LIN {X 0,Y 480.316,Z 788.973,A -85,B 0,C 180,E1 7511.477,E2 7511.477} C_VEL
LIN {X 0,Y 481.888,Z 749.339,A -85,B 0,C 180,E1 7512.908,E2 7512.908} C_VEL
LIN {X 0,Y 449.961,Z 691.44,A -85,B 0,C 180,E1 7518.516,E2 7518.516} C_VEL
LIN {X 0,Y 450.056,Z 691.44,A -85,B 0,C 180,E1 7529.299,E2 7529.299} C_VEL
LIN {X 0,Y 450.366,Z 691.44,A -85,B 0,C 180,E1 7539.308,E2 7539.308} C_VEL
LIN {X 0,Y 450.688,Z 691.44,A -85,B 0,C 180,E1 7549.353,E2 7549.353} C_VEL
LIN {X 0,Y 451.015,Z 691.44,A -85,B 0,C 180,E1 7559.059,E2 7559.059} C_VEL
LIN {X 0,Y 450.905,Z 691.44,A -85,B 0,C 180,E1 7569.708,E2 7569.708} C_VEL
LIN {X 0,Y 451.272,Z 693.873,A -85,B 0,C 180,E1 7570.495,E2 7570.495} C_VEL
LIN {X 0,Y 478.579,Z 746.673,A -85,B 0,C 180,E1 7575.537,E2 7575.537} C_VEL
LIN {X 0,Y 481.013,Z 759.563,A -85,B 0,C 180,E1 7576.393,E2 7576.393} C_VEL
LIN {X 0,Y 473.42,Z 824.079,A -85,B 0,C 180,E1 7580.014,E2 7580.014} C_VEL
LIN {X 0,Y 464.828,Z 880.115,A -85,B 0,C 180,E1 7585.277,E2 7585.277} C_VEL
LIN {X 0,Y 457.425,Z 928.806,A -85,B 0,C 180,E1 7592.429,E2 7592.429} C_VEL
LIN {X 0,Y 453.01,Z 964.235,A -85,B 0,C 180,E1 7600.513,E2 7600.513} C_VEL
LIN {X 0,Y 451.297,Z 983.991,A -85,B 0,C 180,E1 7608.117,E2 7608.117} C_VEL
LIN {X 0,Y 450.543,Z 992.725,A -85,B 0,C 180,E1 7616.237,E2 7616.237} C_VEL
LIN {X 0,Y 451.09,Z 989.426,A -85,B 0,C 180,E1 7624.147,E2 7624.147} C_VEL
LIN {X 0,Y 452.471,Z 971.841,A -85,B 0,C 180,E1 7632.949,E2 7632.949} C_VEL
LIN {X 0,Y 455.599,Z 939.796,A -85,B 0,C 180,E1 7641.38,E2 7641.38} C_VEL
LIN {X 0,Y 462.546,Z 894.419,A -85,B 0,C 180,E1 7648.826,E2 7648.826} C_VEL
LIN {X 0,Y 471.111,Z 840.184,A -85,B 0,C 180,E1 7654.62,E2 7654.62} C_VEL
LIN {X 0,Y 479.119,Z 776.379,A -85,B 0,C 180,E1 7658.798,E2 7658.798} C_VEL
LIN {X 0,Y 480.222,Z 748.401,A -85,B 0,C 180,E1 7660.124,E2 7660.124} C_VEL
LIN {X 0,Y 450.704,Z 691.44,A -85,B 0,C 180,E1 7665.682,E2 7665.682} C_VEL
LIN {X 0,Y 450.338,Z 691.44,A -85,B 0,C 180,E1 7674.914,E2 7674.914} C_VEL
LIN {X 0,Y 449.921,Z 691.44,A -85,B 0,C 180,E1 7684.252,E2 7684.252} C_VEL
LIN {X 0,Y 449.961,Z 691.44,A -85,B 0,C 180,E1 7693.743,E2 7693.743} C_VEL
LIN {X 0,Y 449.854,Z 691.44,A -85,B 0,C 180,E1 7703.8,E2 7703.8} C_VEL
LIN {X 0,Y 450.191,Z 691.44,A -85,B 0,C 180,E1 7713.295,E2 7713.295} C_VEL
LIN {X 0,Y 450.987,Z 691.44,A -85,B 0,C 180,E1 7725.362,E2 7725.362} C_VEL
LIN {X 0,Y 451.028,Z 691.44,A -85,B 0,C 180,E1 7735.153,E2 7735.153} C_VEL
LIN {X 0,Y 451.105,Z 691.44,A -85,B 0,C 180,E1 7742.869,E2 7742.869} C_VEL
LIN {X 0,Y 450.691,Z 691.44,A -85,B 0,C 180,E1 7752.617,E2 7752.617} C_VEL
LIN {X 0,Y 450.376,Z 691.44,A -85,B 0,C 180,E1 7762.769,E2 7762.769} C_VEL
LIN {X 0,Y 450.042,Z 691.44,A -85,B 0,C 180,E1 7771.477,E2 7771.477} C_VEL
LIN {X 0,Y 450.162,Z 693.331,A -85,B 0,C 180,E1 7781.862,E2 7781.862} C_VEL
LIN {X 0,Y 483.134,Z 752.334,A -85,B 0,C 180,E1 7787.26,E2 7787.26} C_VEL
LIN {X 0,Y 477.738,Z 816.415,A -85,B 0,C 180,E1 7789.779,E2 7789.779} C_VEL
LIN {X 0,Y 469.365,Z 878.521,A -85,B 0,C 180,E1 7794.164,E2 7794.164} C_VEL
LIN {X 0,Y 468.241,Z 886.122,A -85,B 0,C 180,E1 7794.871,E2 7794.871} C_VEL
LIN {X 0,Y 457.024,Z 913.577,A -85,B 0,C 180,E1 7797.294,E2 7797.294} C_VEL
LIN {X 0,Y 449.765,Z 960.326,A -85,B 0,C 180,E1 7804.307,E2 7804.307} C_VEL
LIN {X 0,Y 445.009,Z 995.719,A -85,B 0,C 180,E1 7812.691,E2 7812.691} C_VEL
LIN {X 0,Y 443.149,Z 1015.884,A -85,B 0,C 180,E1 7821.134,E2 7821.134} C_VEL
LIN {X 0,Y 442.869,Z 1022.836,A -85,B 0,C 180,E1 7829.017,E2 7829.017} C_VEL
LIN {X 0,Y 443.349,Z 1018.684,A -85,B 0,C 180,E1 7836.88,E2 7836.88} C_VEL
LIN {X 0,Y 444.601,Z 1000.182,A -85,B 0,C 180,E1 7845.846,E2 7845.846} C_VEL
LIN {X 0,Y 448.349,Z 967.674,A -85,B 0,C 180,E1 7854.28,E2 7854.28} C_VEL
LIN {X 0,Y 455.186,Z 924.286,A -85,B 0,C 180,E1 7861.341,E2 7861.341} C_VEL
LIN {X 0,Y 464.152,Z 867.494,A -85,B 0,C 180,E1 7867.331,E2 7867.331} C_VEL
LIN {X 0,Y 472.707,Z 801.444,A -85,B 0,C 180,E1 7871.569,E2 7871.569} C_VEL
LIN {X 0,Y 475.718,Z 752.484,A -85,B 0,C 180,E1 7873.469,E2 7873.469} C_VEL
LIN {X 0,Y 443.691,Z 696.419,A -85,B 0,C 180,E1 7878.995,E2 7878.995} C_VEL
LIN {X 0,Y 441.936,Z 691.44,A -85,B 0,C 180,E1 7879.576,E2 7879.576} C_VEL
LIN {X 0,Y 442.035,Z 691.44,A -85,B 0,C 180,E1 7890.179,E2 7890.179} C_VEL
LIN {X 0,Y 442.406,Z 691.44,A -85,B 0,C 180,E1 7901.01,E2 7901.01} C_VEL
LIN {X 0,Y 442.802,Z 691.44,A -85,B 0,C 180,E1 7911.153,E2 7911.153} C_VEL
LIN {X 0,Y 443.542,Z 691.44,A -85,B 0,C 180,E1 7921.003,E2 7921.003} C_VEL
LIN {X 0,Y 443.012,Z 692.481,A -85,B 0,C 180,E1 7929.261,E2 7929.261} C_VEL
LIN {X 0,Y 471.363,Z 747.296,A -85,B 0,C 180,E1 7934.765,E2 7934.765} C_VEL
LIN {X 0,Y 474.779,Z 761.729,A -85,B 0,C 180,E1 7935.841,E2 7935.841} C_VEL
LIN {X 0,Y 466.841,Z 825.244,A -85,B 0,C 180,E1 7939.475,E2 7939.475} C_VEL
LIN {X 0,Y 457.627,Z 881.883,A -85,B 0,C 180,E1 7944.912,E2 7944.912} C_VEL
LIN {X 0,Y 450.08,Z 928.17,A -85,B 0,C 180,E1 7951.859,E2 7951.859} C_VEL
LIN {X 0,Y 445.374,Z 963.375,A -85,B 0,C 180,E1 7959.945,E2 7959.945} C_VEL
LIN {X 0,Y 443.29,Z 984.327,A -85,B 0,C 180,E1 7968.121,E2 7968.121} C_VEL
LIN {X 0,Y 442.576,Z 992.432,A -85,B 0,C 180,E1 7975.544,E2 7975.544} C_VEL
LIN {X 0,Y 442.986,Z 990.028,A -85,B 0,C 180,E1 7983.678,E2 7983.678} C_VEL
LIN {X 0,Y 444.322,Z 974.867,A -85,B 0,C 180,E1 7992.099,E2 7992.099} C_VEL
LIN {X 0,Y 447.531,Z 944.098,A -85,B 0,C 180,E1 8000.863,E2 8000.863} C_VEL
LIN {X 0,Y 454.538,Z 900.358,A -85,B 0,C 180,E1 8008.566,E2 8008.566} C_VEL
LIN {X 0,Y 463.52,Z 846.298,A -85,B 0,C 180,E1 8014.696,E2 8014.696} C_VEL
LIN {X 0,Y 471.971,Z 784.847,A -85,B 0,C 180,E1 8019.019,E2 8019.019} C_VEL
LIN {X 0,Y 474.063,Z 751.552,A -85,B 0,C 180,E1 8020.649,E2 8020.649} C_VEL
LIN {X 0,Y 444.766,Z 696.762,A -85,B 0,C 180,E1 8026.198,E2 8026.198} C_VEL
LIN {X 0,Y 442.62,Z 691.44,A -85,B 0,C 180,E1 8026.945,E2 8026.945} C_VEL
LIN {X 0,Y 442.17,Z 691.44,A -85,B 0,C 180,E1 8037.604,E2 8037.604} C_VEL
LIN {X 0,Y 441.876,Z 691.44,A -85,B 0,C 180,E1 8046.944,E2 8046.944} C_VEL
LIN {X 0,Y 441.865,Z 691.44,A -85,B 0,C 180,E1 8057.598,E2 8057.598} C_VEL
LIN {X 0,Y 441.942,Z 691.44,A -85,B 0,C 180,E1 8067.824,E2 8067.824} C_VEL
LIN {X 0,Y 441.943,Z 691.44,A -85,B 0,C 180,E1 8076.722,E2 8076.722} C_VEL
LIN {X 0,Y 442.985,Z 691.44,A -85,B 0,C 180,E1 8087.522,E2 8087.522} C_VEL
LIN {X 0,Y 442.874,Z 691.44,A -85,B 0,C 180,E1 8097.032,E2 8097.032} C_VEL
LIN {X 0,Y 442.823,Z 691.44,A -85,B 0,C 180,E1 8104.891,E2 8104.891} C_VEL
LIN {X 0,Y 442.651,Z 691.44,A -85,B 0,C 180,E1 8114.873,E2 8114.873} C_VEL
LIN {X 0,Y 442.244,Z 691.44,A -85,B 0,C 180,E1 8125.369,E2 8125.369} C_VEL
LIN {X 0,Y 441.864,Z 691.44,A -85,B 0,C 180,E1 8136.184,E2 8136.184} C_VEL
LIN {X 0,Y 442.068,Z 692.886,A -85,B 0,C 180,E1 8140.727,E2 8140.727} C_VEL
LIN {X 0,Y 477.127,Z 755.611,A -85,B 0,C 180,E1 8146.717,E2 8146.717} C_VEL
LIN {X 0,Y 470.984,Z 819.692,A -85,B 0,C 180,E1 8149.346,E2 8149.346} C_VEL
LIN {X 0,Y 462.201,Z 881.081,A -85,B 0,C 180,E1 8153.828,E2 8153.828} C_VEL
LIN {X 0,Y 457.024,Z 913.577,A -85,B 0,C 180,E1 8157.294,E2 8157.294} C_VEL
LIN {X 0,Y 445.427,Z 938.536,A -85,B 0,C 180,E1 8160.146,E2 8160.146} C_VEL
LIN {X 0,Y 438.993,Z 978.351,A -85,B 0,C 180,E1 8167.649,E2 8167.649} C_VEL
LIN {X 0,Y 435.805,Z 1004.335,A -85,B 0,C 180,E1 8175.376,E2 8175.376} C_VEL
LIN {X 0,Y 435.111,Z 1019.184,A -85,B 0,C 180,E1 8183.405,E2 8183.405} C_VEL
LIN {X 0,Y 435.328,Z 1022.837,A -85,B 0,C 180,E1 8190.998,E2 8190.998} C_VEL
LIN {X 0,Y 435.348,Z 1015.887,A -85,B 0,C 180,E1 8199.024,E2 8199.024} C_VEL
LIN {X 0,Y 436.853,Z 995.72,A -85,B 0,C 180,E1 8207.642,E2 8207.642} C_VEL
LIN {X 0,Y 441.383,Z 962.92,A -85,B 0,C 180,E1 8215.667,E2 8215.667} C_VEL
LIN {X 0,Y 449.416,Z 915.357,A -85,B 0,C 180,E1 8222.997,E2 8222.997} C_VEL
LIN {X 0,Y 459.194,Z 856.838,A -85,B 0,C 180,E1 8228.769,E2 8228.769} C_VEL
LIN {X 0,Y 467.619,Z 792.407,A -85,B 0,C 180,E1 8232.591,E2 8232.591} C_VEL
LIN {X 0,Y 469.538,Z 755.476,A -85,B 0,C 180,E1 8234.06,E2 8234.06} C_VEL
LIN {X 0,Y 437.3,Z 697.979,A -85,B 0,C 180,E1 8239.937,E2 8239.937} C_VEL
LIN {X 0,Y 433.861,Z 691.44,A -85,B 0,C 180,E1 8240.866,E2 8240.866} C_VEL
LIN {X 0,Y 434.008,Z 691.44,A -85,B 0,C 180,E1 8251.866,E2 8251.866} C_VEL
LIN {X 0,Y 434.438,Z 691.44,A -85,B 0,C 180,E1 8262.756,E2 8262.756} C_VEL
LIN {X 0,Y 435.03,Z 691.44,A -85,B 0,C 180,E1 8273.826,E2 8273.826} C_VEL
LIN {X 0,Y 435.092,Z 691.44,A -85,B 0,C 180,E1 8283.021,E2 8283.021} C_VEL
LIN {X 0,Y 435.012,Z 692.594,A -85,B 0,C 180,E1 8288.011,E2 8288.011} C_VEL
LIN {X 0,Y 463.641,Z 746.298,A -85,B 0,C 180,E1 8293.815,E2 8293.815} C_VEL
LIN {X 0,Y 468.572,Z 764.043,A -85,B 0,C 180,E1 8295.283,E2 8295.283} C_VEL
LIN {X 0,Y 460.152,Z 827.524,A -85,B 0,C 180,E1 8299.004,E2 8299.004} C_VEL
LIN {X 0,Y 450.443,Z 883.623,A -85,B 0,C 180,E1 8304.532,E2 8304.532} C_VEL
LIN {X 0,Y 442.524,Z 928.985,A -85,B 0,C 180,E1 8311.512,E2 8311.512} C_VEL
LIN {X 0,Y 437.377,Z 964.49,A -85,B 0,C 180,E1 8319.952,E2 8319.952} C_VEL
LIN {X 0,Y 435.145,Z 985.382,A -85,B 0,C 180,E1 8328.594,E2 8328.594} C_VEL
LIN {X 0,Y 434.43,Z 992.899,A -85,B 0,C 180,E1 8337.218,E2 8337.218} C_VEL
LIN {X 0,Y 435.302,Z 987.95,A -85,B 0,C 180,E1 8345.566,E2 8345.566} C_VEL
LIN {X 0,Y 436.609,Z 969.298,A -85,B 0,C 180,E1 8354.415,E2 8354.415} C_VEL
LIN {X 0,Y 440.765,Z 937.007,A -85,B 0,C 180,E1 8362.831,E2 8362.831} C_VEL
LIN {X 0,Y 448.707,Z 892.747,A -85,B 0,C 180,E1 8370.193,E2 8370.193} C_VEL
LIN {X 0,Y 458.535,Z 837.577,A -85,B 0,C 180,E1 8376.074,E2 8376.074} C_VEL
LIN {X 0,Y 467.265,Z 774.86,A -85,B 0,C 180,E1 8380.164,E2 8380.164} C_VEL
LIN {X 0,Y 467.82,Z 754.567,A -85,B 0,C 180,E1 8381.207,E2 8381.207} C_VEL
LIN {X 0,Y 437.999,Z 697.971,A -85,B 0,C 180,E1 8387.129,E2 8387.129} C_VEL
LIN {X 0,Y 434.482,Z 691.44,A -85,B 0,C 180,E1 8388.218,E2 8388.218} C_VEL
LIN {X 0,Y 434.132,Z 691.44,A -85,B 0,C 180,E1 8398.16,E2 8398.16} C_VEL
LIN {X 0,Y 433.796,Z 691.44,A -85,B 0,C 180,E1 8408.061,E2 8408.061} C_VEL
LIN {X 0,Y 433.777,Z 691.44,A -85,B 0,C 180,E1 8418.782,E2 8418.782} C_VEL
LIN {X 0,Y 433.948,Z 691.44,A -85,B 0,C 180,E1 8429.511,E2 8429.511} C_VEL
LIN {X 0,Y 434.112,Z 691.44,A -85,B 0,C 180,E1 8440.584,E2 8440.584} C_VEL
LIN {X 0,Y 434.8,Z 691.44,A -85,B 0,C 180,E1 8448.912,E2 8448.912} C_VEL
LIN {X 0,Y 435.028,Z 691.44,A -85,B 0,C 180,E1 8458.978,E2 8458.978} C_VEL
LIN {X 0,Y 434.915,Z 691.44,A -85,B 0,C 180,E1 8469.008,E2 8469.008} C_VEL
LIN {X 0,Y 434.413,Z 691.44,A -85,B 0,C 180,E1 8479.353,E2 8479.353} C_VEL
LIN {X 0,Y 433.951,Z 691.44,A -85,B 0,C 180,E1 8490.435,E2 8490.435} C_VEL
LIN {X 0,Y 433.98,Z 692.906,A -85,B 0,C 180,E1 8499.538,E2 8499.538} C_VEL
LIN {X 0,Y 469.785,Z 755.903,A -85,B 0,C 180,E1 8505.908,E2 8505.908} C_VEL
LIN {X 0,Y 464.007,Z 825.434,A -85,B 0,C 180,E1 8509.049,E2 8509.049} C_VEL
LIN {X 0,Y 454.85,Z 884.36,A -85,B 0,C 180,E1 8513.567,E2 8513.567} C_VEL
LIN {X 0,Y 445.427,Z 938.536,A -85,B 0,C 180,E1 8520.146,E2 8520.146} C_VEL
LIN {X 0,Y 434.591,Z 960.584,A -85,B 0,C 180,E1 8523.488,E2 8523.488} C_VEL
LIN {X 0,Y 429.699,Z 993.822,A -85,B 0,C 180,E1 8531.466,E2 8531.466} C_VEL
LIN {X 0,Y 427.566,Z 1014.284,A -85,B 0,C 180,E1 8539.777,E2 8539.777} C_VEL
LIN {X 0,Y 427.102,Z 1022.147,A -85,B 0,C 180,E1 8546.944,E2 8546.944} C_VEL
LIN {X 0,Y 427.09,Z 1020.767,A -85,B 0,C 180,E1 8555.096,E2 8555.096} C_VEL
LIN {X 0,Y 428.058,Z 1006.922,A -85,B 0,C 180,E1 8563.845,E2 8563.845} C_VEL
LIN {X 0,Y 431.905,Z 978.304,A -85,B 0,C 180,E1 8572.736,E2 8572.736} C_VEL
LIN {X 0,Y 438.801,Z 935.959,A -85,B 0,C 180,E1 8580.671,E2 8580.671} C_VEL
LIN {X 0,Y 448.42,Z 881.102,A -85,B 0,C 180,E1 8587.297,E2 8587.297} C_VEL
LIN {X 0,Y 458.32,Z 817.471,A -85,B 0,C 180,E1 8592.018,E2 8592.018} C_VEL
LIN {X 0,Y 463.461,Z 758.843,A -85,B 0,C 180,E1 8594.624,E2 8594.624} C_VEL
LIN {X 0,Y 433.366,Z 704.271,A -85,B 0,C 180,E1 8600.399,E2 8600.399} C_VEL
LIN {X 0,Y 425.796,Z 691.44,A -85,B 0,C 180,E1 8602.436,E2 8602.436} C_VEL
LIN {X 0,Y 425.989,Z 691.44,A -85,B 0,C 180,E1 8613.59,E2 8613.59} C_VEL
LIN {X 0,Y 426.53,Z 691.44,A -85,B 0,C 180,E1 8624.551,E2 8624.551} C_VEL
LIN {X 0,Y 427.063,Z 691.44,A -85,B 0,C 180,E1 8634.928,E2 8634.928} C_VEL
LIN {X 0,Y 427.076,Z 691.44,A -85,B 0,C 180,E1 8643.078,E2 8643.078} C_VEL
LIN {X 0,Y 427.165,Z 693.273,A -85,B 0,C 180,E1 8646.701,E2 8646.701} C_VEL
LIN {X 0,Y 455.681,Z 744.692,A -85,B 0,C 180,E1 8652.763,E2 8652.763} C_VEL
LIN {X 0,Y 462.28,Z 767.632,A -85,B 0,C 180,E1 8654.764,E2 8654.764} C_VEL
LIN {X 0,Y 453.428,Z 830.232,A -85,B 0,C 180,E1 8658.558,E2 8658.558} C_VEL
LIN {X 0,Y 443.065,Z 886.375,A -85,B 0,C 180,E1 8664.262,E2 8664.262} C_VEL
LIN {X 0,Y 434.613,Z 932.02,A -85,B 0,C 180,E1 8671.565,E2 8671.565} C_VEL
LIN {X 0,Y 429.081,Z 967.243,A -85,B 0,C 180,E1 8680.5,E2 8680.5} C_VEL
LIN {X 0,Y 427.068,Z 986.144,A -85,B 0,C 180,E1 8688.899,E2 8688.899} C_VEL
LIN {X 0,Y 426.417,Z 992.838,A -85,B 0,C 180,E1 8696.778,E2 8696.778} C_VEL
LIN {X 0,Y 427.17,Z 988.895,A -85,B 0,C 180,E1 8704.974,E2 8704.974} C_VEL
LIN {X 0,Y 428.67,Z 970.876,A -85,B 0,C 180,E1 8714.152,E2 8714.152} C_VEL
LIN {X 0,Y 433.006,Z 938.815,A -85,B 0,C 180,E1 8722.955,E2 8722.955} C_VEL
LIN {X 0,Y 441.315,Z 895.135,A -85,B 0,C 180,E1 8730.46,E2 8730.46} C_VEL
LIN {X 0,Y 451.732,Z 840.037,A -85,B 0,C 180,E1 8736.517,E2 8736.517} C_VEL
LIN {X 0,Y 461.007,Z 776.696,A -85,B 0,C 180,E1 8740.751,E2 8740.751} C_VEL
LIN {X 0,Y 461.604,Z 757.462,A -85,B 0,C 180,E1 8741.786,E2 8741.786} C_VEL
LIN {X 0,Y 433.132,Z 703.469,A -85,B 0,C 180,E1 8747.708,E2 8747.708} C_VEL
LIN {X 0,Y 426.486,Z 691.44,A -85,B 0,C 180,E1 8749.413,E2 8749.413} C_VEL
LIN {X 0,Y 426.005,Z 691.44,A -85,B 0,C 180,E1 8759.193,E2 8759.193} C_VEL
LIN {X 0,Y 425.776,Z 691.44,A -85,B 0,C 180,E1 8769.955,E2 8769.955} C_VEL
LIN {X 0,Y 425.703,Z 691.44,A -85,B 0,C 180,E1 8780.038,E2 8780.038} C_VEL
LIN {X 0,Y 425.919,Z 691.44,A -85,B 0,C 180,E1 8790.806,E2 8790.806} C_VEL
LIN {X 0,Y 426.4,Z 691.44,A -85,B 0,C 180,E1 8802.371,E2 8802.371} C_VEL
LIN {X 0,Y 426.759,Z 691.44,A -85,B 0,C 180,E1 8810.77,E2 8810.77} C_VEL
LIN {X 0,Y 427.532,Z 691.44,A -85,B 0,C 180,E1 8820.993,E2 8820.993} C_VEL
LIN {X 0,Y 426.643,Z 691.44,A -85,B 0,C 180,E1 8831.984,E2 8831.984} C_VEL
LIN {X 0,Y 426.276,Z 691.44,A -85,B 0,C 180,E1 8841.92,E2 8841.92} C_VEL
LIN {X 0,Y 425.848,Z 691.44,A -85,B 0,C 180,E1 8853.124,E2 8853.124} C_VEL
LIN {X 0,Y 425.888,Z 692.826,A -85,B 0,C 180,E1 8858.288,E2 8858.288} C_VEL
LIN {X 0,Y 461.677,Z 754.671,A -85,B 0,C 180,E1 8864.925,E2 8864.925} C_VEL
LIN {X 0,Y 464.446,Z 765.843,A -85,B 0,C 180,E1 8865.694,E2 8865.694} C_VEL
LIN {X 0,Y 456.858,Z 831.45,A -85,B 0,C 180,E1 8868.769,E2 8868.769} C_VEL
LIN {X 0,Y 446.862,Z 891.455,A -85,B 0,C 180,E1 8873.692,E2 8873.692} C_VEL
LIN {X 0,Y 437.185,Z 943.235,A -85,B 0,C 180,E1 8880.411,E2 8880.411} C_VEL
LIN {X 0,Y 434.591,Z 960.584,A -85,B 0,C 180,E1 8883.488,E2 8883.488} C_VEL
LIN {X 0,Y 423.344,Z 979.641,A -85,B 0,C 180,E1 8887.201,E2 8887.201} C_VEL
LIN {X 0,Y 419.88,Z 1005.674,A -85,B 0,C 180,E1 8895.344,E2 8895.344} C_VEL
LIN {X 0,Y 419.053,Z 1018.681,A -85,B 0,C 180,E1 8902.717,E2 8902.717} C_VEL
LIN {X 0,Y 419.324,Z 1022.836,A -85,B 0,C 180,E1 8911.036,E2 8911.036} C_VEL
LIN {X 0,Y 419.329,Z 1015.887,A -85,B 0,C 180,E1 8919.372,E2 8919.372} C_VEL
LIN {X 0,Y 420.979,Z 997.105,A -85,B 0,C 180,E1 8927.842,E2 8927.842} C_VEL
LIN {X 0,Y 425.691,Z 965.859,A -85,B 0,C 180,E1 8935.895,E2 8935.895} C_VEL
LIN {X 0,Y 434.736,Z 917.907,A -85,B 0,C 180,E1 8943.742,E2 8943.742} C_VEL
LIN {X 0,Y 445.413,Z 860.946,A -85,B 0,C 180,E1 8949.672,E2 8949.672} C_VEL
LIN {X 0,Y 454.871,Z 798.066,A -85,B 0,C 180,E1 8953.673,E2 8953.673} C_VEL
LIN {X 0,Y 457.316,Z 762.072,A -85,B 0,C 180,E1 8955.222,E2 8955.222} C_VEL
LIN {X 0,Y 429.354,Z 710.276,A -85,B 0,C 180,E1 8960.9,E2 8960.9} C_VEL
LIN {X 0,Y 417.753,Z 691.44,A -85,B 0,C 180,E1 8963.643,E2 8963.643} C_VEL
LIN {X 0,Y 417.91,Z 691.44,A -85,B 0,C 180,E1 8973.039,E2 8973.039} C_VEL
LIN {X 0,Y 418.473,Z 691.44,A -85,B 0,C 180,E1 8984.246,E2 8984.246} C_VEL
LIN {X 0,Y 419.058,Z 691.44,A -85,B 0,C 180,E1 8994.831,E2 8994.831} C_VEL
LIN {X 0,Y 419.059,Z 691.44,A -85,B 0,C 180,E1 9003.137,E2 9003.137} C_VEL
LIN {X 0,Y 419.116,Z 693.418,A -85,B 0,C 180,E1 9005.217,E2 9005.217} C_VEL
LIN {X 0,Y 446.817,Z 741.093,A -85,B 0,C 180,E1 9011.431,E2 9011.431} C_VEL
LIN {X 0,Y 456.159,Z 769.764,A -85,B 0,C 180,E1 9014.161,E2 9014.161} C_VEL
LIN {X 0,Y 446.969,Z 831.246,A -85,B 0,C 180,E1 9017.965,E2 9017.965} C_VEL
LIN {X 0,Y 435.782,Z 888.817,A -85,B 0,C 180,E1 9023.944,E2 9023.944} C_VEL
LIN {X 0,Y 426.809,Z 934.302,A -85,B 0,C 180,E1 9031.487,E2 9031.487} C_VEL
LIN {X 0,Y 421.196,Z 967.832,A -85,B 0,C 180,E1 9040.36,E2 9040.36} C_VEL
LIN {X 0,Y 419.057,Z 986.495,A -85,B 0,C 180,E1 9048.952,E2 9048.952} C_VEL
LIN {X 0,Y 418.411,Z 992.591,A -85,B 0,C 180,E1 9055.794,E2 9055.794} C_VEL
LIN {X 0,Y 419.044,Z 989.581,A -85,B 0,C 180,E1 9064.454,E2 9064.454} C_VEL
LIN {X 0,Y 420.638,Z 973.055,A -85,B 0,C 180,E1 9073.659,E2 9073.659} C_VEL
LIN {X 0,Y 425.032,Z 941.706,A -85,B 0,C 180,E1 9082.822,E2 9082.822} C_VEL
LIN {X 0,Y 433.698,Z 898.635,A -85,B 0,C 180,E1 9090.582,E2 9090.582} C_VEL
LIN {X 0,Y 444.661,Z 843.705,A -85,B 0,C 180,E1 9096.861,E2 9096.861} C_VEL
LIN {X 0,Y 454.309,Z 782.08,A -85,B 0,C 180,E1 9101.17,E2 9101.17} C_VEL
LIN {X 0,Y 455.739,Z 761.278,A -85,B 0,C 180,E1 9102.289,E2 9102.289} C_VEL
LIN {X 0,Y 428.351,Z 708.711,A -85,B 0,C 180,E1 9108.276,E2 9108.276} C_VEL
LIN {X 0,Y 418.332,Z 691.44,A -85,B 0,C 180,E1 9110.689,E2 9110.689} C_VEL
LIN {X 0,Y 417.907,Z 691.44,A -85,B 0,C 180,E1 9121.774,E2 9121.774} C_VEL
LIN {X 0,Y 417.79,Z 691.44,A -85,B 0,C 180,E1 9132.223,E2 9132.223} C_VEL
LIN {X 0,Y 417.67,Z 691.44,A -85,B 0,C 180,E1 9143.145,E2 9143.145} C_VEL
LIN {X 0,Y 417.938,Z 691.44,A -85,B 0,C 180,E1 9152.986,E2 9152.986} C_VEL
LIN {X 0,Y 418.687,Z 691.44,A -85,B 0,C 180,E1 9164.205,E2 9164.205} C_VEL
LIN {X 0,Y 419.031,Z 691.44,A -85,B 0,C 180,E1 9174.858,E2 9174.858} C_VEL
LIN {X 0,Y 419.049,Z 691.44,A -85,B 0,C 180,E1 9183.089,E2 9183.089} C_VEL
LIN {X 0,Y 418.579,Z 691.44,A -85,B 0,C 180,E1 9193.603,E2 9193.603} C_VEL
LIN {X 0,Y 418.167,Z 691.44,A -85,B 0,C 180,E1 9204.635,E2 9204.635} C_VEL
LIN {X 0,Y 417.667,Z 691.44,A -85,B 0,C 180,E1 9215.159,E2 9215.159} C_VEL
LIN {X 0,Y 418.026,Z 693.601,A -85,B 0,C 180,E1 9217.019,E2 9217.019} C_VEL
LIN {X 0,Y 454.384,Z 754.819,A -85,B 0,C 180,E1 9224.041,E2 9224.041} C_VEL
LIN {X 0,Y 458.366,Z 768.472,A -85,B 0,C 180,E1 9225.09,E2 9225.09} C_VEL
LIN {X 0,Y 450.191,Z 834.018,A -85,B 0,C 180,E1 9228.28,E2 9228.28} C_VEL
LIN {X 0,Y 439.643,Z 894.023,A -85,B 0,C 180,E1 9233.364,E2 9233.364} C_VEL
LIN {X 0,Y 429.15,Z 947.304,A -85,B 0,C 180,E1 9240.591,E2 9240.591} C_VEL
LIN {X 0,Y 423.344,Z 979.641,A -85,B 0,C 180,E1 9247.201,E2 9247.201} C_VEL
LIN {X 0,Y 413.761,Z 995.482,A -85,B 0,C 180,E1 9251.357,E2 9251.357} C_VEL
LIN {X 0,Y 411.336,Z 1015.884,A -85,B 0,C 180,E1 9260.442,E2 9260.442} C_VEL
LIN {X 0,Y 410.909,Z 1022.836,A -85,B 0,C 180,E1 9268.941,E2 9268.941} C_VEL
LIN {X 0,Y 411.422,Z 1018.684,A -85,B 0,C 180,E1 9277.417,E2 9277.417} C_VEL
LIN {X 0,Y 412.833,Z 1001.048,A -85,B 0,C 180,E1 9286.726,E2 9286.726} C_VEL
LIN {X 0,Y 417.538,Z 969.183,A -85,B 0,C 180,E1 9295.569,E2 9295.569} C_VEL
LIN {X 0,Y 426.41,Z 923.933,A -85,B 0,C 180,E1 9303.479,E2 9303.479} C_VEL
LIN {X 0,Y 437.763,Z 867.701,A -85,B 0,C 180,E1 9309.75,E2 9309.75} C_VEL
LIN {X 0,Y 448.119,Z 803.225,A -85,B 0,C 180,E1 9314.119,E2 9314.119} C_VEL
LIN {X 0,Y 451.313,Z 765.282,A -85,B 0,C 180,E1 9315.827,E2 9315.827} C_VEL
LIN {X 0,Y 424.712,Z 715.308,A -85,B 0,C 180,E1 9321.554,E2 9321.554} C_VEL
LIN {X 0,Y 409.697,Z 691.44,A -85,B 0,C 180,E1 9325.388,E2 9325.388} C_VEL
LIN {X 0,Y 410.022,Z 691.44,A -85,B 0,C 180,E1 9335.065,E2 9335.065} C_VEL
LIN {X 0,Y 410.56,Z 691.44,A -85,B 0,C 180,E1 9346.127,E2 9346.127} C_VEL
LIN {X 0,Y 410.891,Z 691.44,A -85,B 0,C 180,E1 9356.849,E2 9356.849} C_VEL
LIN {X 0,Y 411.175,Z 693.115,A -85,B 0,C 180,E1 9363.582,E2 9363.582} C_VEL
LIN {X 0,Y 438.442,Z 738.988,A -85,B 0,C 180,E1 9370.137,E2 9370.137} C_VEL
LIN {X 0,Y 450.041,Z 772.612,A -85,B 0,C 180,E1 9373.573,E2 9373.573} C_VEL
LIN {X 0,Y 440.195,Z 834.426,A -85,B 0,C 180,E1 9377.539,E2 9377.539} C_VEL
LIN {X 0,Y 428.549,Z 890.967,A -85,B 0,C 180,E1 9383.591,E2 9383.591} C_VEL
LIN {X 0,Y 419.071,Z 936.108,A -85,B 0,C 180,E1 9391.306,E2 9391.306} C_VEL
LIN {X 0,Y 413.19,Z 969.123,A -85,B 0,C 180,E1 9400.379,E2 9400.379} C_VEL
LIN {X 0,Y 411.036,Z 987.104,A -85,B 0,C 180,E1 9409.211,E2 9409.211} C_VEL
LIN {X 0,Y 410.28,Z 992.952,A -85,B 0,C 180,E1 9417.566,E2 9417.566} C_VEL
LIN {X 0,Y 411.25,Z 987.898,A -85,B 0,C 180,E1 9426.052,E2 9426.052} C_VEL
LIN {X 0,Y 412.83,Z 970.292,A -85,B 0,C 180,E1 9435.09,E2 9435.09} C_VEL
LIN {X 0,Y 417.872,Z 939.987,A -85,B 0,C 180,E1 9443.746,E2 9443.746} C_VEL
LIN {X 0,Y 427.273,Z 896.344,A -85,B 0,C 180,E1 9451.527,E2 9451.527} C_VEL
LIN {X 0,Y 438.713,Z 841.925,A -85,B 0,C 180,E1 9457.704,E2 9457.704} C_VEL
LIN {X 0,Y 449.03,Z 778.181,A -85,B 0,C 180,E1 9462.072,E2 9462.072} C_VEL
LIN {X 0,Y 449.408,Z 764.01,A -85,B 0,C 180,E1 9462.908,E2 9462.908} C_VEL
LIN {X 0,Y 422.014,Z 710.772,A -85,B 0,C 180,E1 9469.206,E2 9469.206} C_VEL
LIN {X 0,Y 410.303,Z 691.44,A -85,B 0,C 180,E1 9471.955,E2 9471.955} C_VEL
LIN {X 0,Y 409.785,Z 691.44,A -85,B 0,C 180,E1 9482.48,E2 9482.48} C_VEL
LIN {X 0,Y 409.664,Z 691.44,A -85,B 0,C 180,E1 9493.728,E2 9493.728} C_VEL
LIN {X 0,Y 409.693,Z 691.44,A -85,B 0,C 180,E1 9504.939,E2 9504.939} C_VEL
LIN {X 0,Y 409.928,Z 691.44,A -85,B 0,C 180,E1 9515.098,E2 9515.098} C_VEL
LIN {X 0,Y 410.827,Z 691.44,A -85,B 0,C 180,E1 9526.085,E2 9526.085} C_VEL
LIN {X 0,Y 410.895,Z 691.44,A -85,B 0,C 180,E1 9536.8,E2 9536.8} C_VEL
LIN {X 0,Y 410.822,Z 691.44,A -85,B 0,C 180,E1 9545.273,E2 9545.273} C_VEL
LIN {X 0,Y 410.495,Z 691.44,A -85,B 0,C 180,E1 9556.068,E2 9556.068} C_VEL
LIN {X 0,Y 409.957,Z 691.44,A -85,B 0,C 180,E1 9567.528,E2 9567.528} C_VEL
LIN {X 0,Y 409.818,Z 693.069,A -85,B 0,C 180,E1 9575.579,E2 9575.579} C_VEL
LIN {X 0,Y 446.604,Z 754.26,A -85,B 0,C 180,E1 9583.032,E2 9583.032} C_VEL
LIN {X 0,Y 452.348,Z 770.885,A -85,B 0,C 180,E1 9584.465,E2 9584.465} C_VEL
LIN {X 0,Y 443.794,Z 835.154,A -85,B 0,C 180,E1 9587.681,E2 9587.681} C_VEL
LIN {X 0,Y 432.797,Z 894.309,A -85,B 0,C 180,E1 9592.78,E2 9592.78} C_VEL
LIN {X 0,Y 421.727,Z 947.432,A -85,B 0,C 180,E1 9600.112,E2 9600.112} C_VEL
LIN {X 0,Y 414.703,Z 986.351,A -85,B 0,C 180,E1 9608.622,E2 9608.622} C_VEL
LIN {X 0,Y 413.761,Z 995.482,A -85,B 0,C 180,E1 9611.357,E2 9611.357} C_VEL
LIN {X 0,Y 403.82,Z 1007.688,A -85,B 0,C 180,E1 9615.822,E2 9615.822} C_VEL
LIN {X 0,Y 403.309,Z 1020.763,A -85,B 0,C 180,E1 9624.601,E2 9624.601} C_VEL
LIN {X 0,Y 403.187,Z 1022.147,A -85,B 0,C 180,E1 9633.236,E2 9633.236} C_VEL
LIN {X 0,Y 403.42,Z 1012.164,A -85,B 0,C 180,E1 9641.94,E2 9641.94} C_VEL
LIN {X 0,Y 406.406,Z 989.464,A -85,B 0,C 180,E1 9650.777,E2 9650.777} C_VEL
LIN {X 0,Y 413.744,Z 950.864,A -85,B 0,C 180,E1 9659.68,E2 9659.68} C_VEL
LIN {X 0,Y 424.243,Z 901.282,A -85,B 0,C 180,E1 9666.97,E2 9666.97} C_VEL
LIN {X 0,Y 436.304,Z 840.89,A -85,B 0,C 180,E1 9672.549,E2 9672.549} C_VEL
LIN {X 0,Y 445.814,Z 777.518,A -85,B 0,C 180,E1 9675.926,E2 9675.926} C_VEL
LIN {X 0,Y 443.999,Z 765.037,A -85,B 0,C 180,E1 9676.789,E2 9676.789} C_VEL
LIN {X 0,Y 417.569,Z 716.204,A -85,B 0,C 180,E1 9682.833,E2 9682.833} C_VEL
LIN {X 0,Y 401.696,Z 691.44,A -85,B 0,C 180,E1 9687.569,E2 9687.569} C_VEL
LIN {X 0,Y 402.146,Z 691.44,A -85,B 0,C 180,E1 9699.024,E2 9699.024} C_VEL
LIN {X 0,Y 402.677,Z 691.44,A -85,B 0,C 180,E1 9710.264,E2 9710.264} C_VEL
LIN {X 0,Y 403.479,Z 691.44,A -85,B 0,C 180,E1 9721.102,E2 9721.102} C_VEL
LIN {X 0,Y 403.897,Z 694.594,A -85,B 0,C 180,E1 9721.976,E2 9721.976} C_VEL
LIN {X 0,Y 428.98,Z 734.824,A -85,B 0,C 180,E1 9728.458,E2 9728.458} C_VEL
LIN {X 0,Y 444.092,Z 774.606,A -85,B 0,C 180,E1 9732.931,E2 9732.931} C_VEL
LIN {X 0,Y 433.862,Z 835.337,A -85,B 0,C 180,E1 9736.901,E2 9736.901} C_VEL
LIN {X 0,Y 421.865,Z 890.788,A -85,B 0,C 180,E1 9742.9,E2 9742.9} C_VEL
LIN {X 0,Y 411.651,Z 936.75,A -85,B 0,C 180,E1 9750.874,E2 9750.874} C_VEL
LIN {X 0,Y 405.536,Z 969.039,A -85,B 0,C 180,E1 9759.903,E2 9759.903} C_VEL
LIN {X 0,Y 403.127,Z 986.883,A -85,B 0,C 180,E1 9768.793,E2 9768.793} C_VEL
LIN {X 0,Y 402.235,Z 992.984,A -85,B 0,C 180,E1 9778.117,E2 9778.117} C_VEL
LIN {X 0,Y 403.277,Z 986.684,A -85,B 0,C 180,E1 9787.247,E2 9787.247} C_VEL
LIN {X 0,Y 405.096,Z 969.309,A -85,B 0,C 180,E1 9795.907,E2 9795.907} C_VEL
LIN {X 0,Y 410.841,Z 938.262,A -85,B 0,C 180,E1 9804.702,E2 9804.702} C_VEL
LIN {X 0,Y 421.054,Z 893.512,A -85,B 0,C 180,E1 9812.583,E2 9812.583} C_VEL
LIN {X 0,Y 433.057,Z 838.605,A -85,B 0,C 180,E1 9818.693,E2 9818.693} C_VEL
LIN {X 0,Y 443.486,Z 776.886,A -85,B 0,C 180,E1 9822.853,E2 9822.853} C_VEL
LIN {X 0,Y 442.147,Z 764.097,A -85,B 0,C 180,E1 9823.832,E2 9823.832} C_VEL
LIN {X 0,Y 414.707,Z 711.813,A -85,B 0,C 180,E1 9830.376,E2 9830.376} C_VEL
LIN {X 0,Y 402.184,Z 691.44,A -85,B 0,C 180,E1 9833.342,E2 9833.342} C_VEL
LIN {X 0,Y 401.745,Z 691.44,A -85,B 0,C 180,E1 9843.213,E2 9843.213} C_VEL
LIN {X 0,Y 401.6,Z 691.44,A -85,B 0,C 180,E1 9854.355,E2 9854.355} C_VEL
LIN {X 0,Y 401.626,Z 691.44,A -85,B 0,C 180,E1 9864.333,E2 9864.333} C_VEL
LIN {X 0,Y 401.834,Z 691.44,A -85,B 0,C 180,E1 9874.237,E2 9874.237} C_VEL
LIN {X 0,Y 402.762,Z 691.44,A -85,B 0,C 180,E1 9885.801,E2 9885.801} C_VEL
LIN {X 0,Y 402.896,Z 691.44,A -85,B 0,C 180,E1 9896.737,E2 9896.737} C_VEL
LIN {X 0,Y 402.812,Z 691.44,A -85,B 0,C 180,E1 9905.378,E2 9905.378} C_VEL
LIN {X 0,Y 402.466,Z 691.44,A -85,B 0,C 180,E1 9916.397,E2 9916.397} C_VEL
LIN {X 0,Y 401.958,Z 691.44,A -85,B 0,C 180,E1 9927.469,E2 9927.469} C_VEL
LIN {X 0,Y 401.774,Z 692.596,A -85,B 0,C 180,E1 9934.081,E2 9934.081} C_VEL
LIN {X 0,Y 438.914,Z 753.981,A -85,B 0,C 180,E1 9941.995,E2 9941.995} C_VEL
LIN {X 0,Y 446.228,Z 773.751,A -85,B 0,C 180,E1 9943.853,E2 9943.853} C_VEL
LIN {X 0,Y 436.789,Z 840.432,A -85,B 0,C 180,E1 9947.349,E2 9947.349} C_VEL
LIN {X 0,Y 424.936,Z 899.775,A -85,B 0,C 180,E1 9952.779,E2 9952.779} C_VEL
LIN {X 0,Y 413.894,Z 949.75,A -85,B 0,C 180,E1 9960.028,E2 9960.028} C_VEL
LIN {X 0,Y 406.662,Z 988.296,A -85,B 0,C 180,E1 9968.831,E2 9968.831} C_VEL
LIN {X 0,Y 403.82,Z 1007.688,A -85,B 0,C 180,E1 9975.822,E2 9975.822} C_VEL
LIN {X 0,Y 395.291,Z 1016.356,A -85,B 0,C 180,E1 9980.636,E2 9980.636} C_VEL
LIN {X 0,Y 394.928,Z 1022.663,A -85,B 0,C 180,E1 9988.898,E2 9988.898} C_VEL
LIN {X 0,Y 395.433,Z 1018.385,A -85,B 0,C 180,E1 9997.718,E2 9997.718} C_VEL
LIN {X 0,Y 396.946,Z 1001.04,A -85,B 0,C 180,E1 10007.131,E2 10007.131} C_VEL
LIN {X 0,Y 402.165,Z 969.602,A -85,B 0,C 180,E1 10016.319,E2 10016.319} C_VEL
LIN {X 0,Y 412.118,Z 924.763,A -85,B 0,C 180,E1 10024.512,E2 10024.512} C_VEL
LIN {X 0,Y 424.757,Z 868.291,A -85,B 0,C 180,E1 10031.033,E2 10031.033} C_VEL
LIN {X 0,Y 436.189,Z 804.425,A -85,B 0,C 180,E1 10035.498,E2 10035.498} C_VEL
LIN {X 0,Y 439.388,Z 771.385,A -85,B 0,C 180,E1 10037.103,E2 10037.103} C_VEL
LIN {X 0,Y 414.172,Z 722.621,A -85,B 0,C 180,E1 10043.29,E2 10043.29} C_VEL
LIN {X 0,Y 393.738,Z 691.44,A -85,B 0,C 180,E1 10049.467,E2 10049.467} C_VEL
LIN {X 0,Y 394.208,Z 691.44,A -85,B 0,C 180,E1 10060.931,E2 10060.931} C_VEL
LIN {X 0,Y 394.902,Z 691.44,A -85,B 0,C 180,E1 10072.298,E2 10072.298} C_VEL
LIN {X 0,Y 395.321,Z 693.22,A -85,B 0,C 180,E1 10079.682,E2 10079.682} C_VEL
LIN {X 0,Y 420.907,Z 733.174,A -85,B 0,C 180,E1 10087.012,E2 10087.012} C_VEL
LIN {X 0,Y 438.323,Z 775.478,A -85,B 0,C 180,E1 10092.209,E2 10092.209} C_VEL
LIN {X 0,Y 427.391,Z 837.355,A -85,B 0,C 180,E1 10096.338,E2 10096.338} C_VEL
LIN {X 0,Y 414.725,Z 892.676,A -85,B 0,C 180,E1 10102.483,E2 10102.483} C_VEL
LIN {X 0,Y 404.168,Z 937.657,A -85,B 0,C 180,E1 10110.478,E2 10110.478} C_VEL
LIN {X 0,Y 397.636,Z 970.048,A -85,B 0,C 180,E1 10119.812,E2 10119.812} C_VEL
LIN {X 0,Y 395.229,Z 987.03,A -85,B 0,C 180,E1 10128.505,E2 10128.505} C_VEL
LIN {X 0,Y 394.269,Z 992.993,A -85,B 0,C 180,E1 10136.075,E2 10136.075} C_VEL
LIN {X 0,Y 395.027,Z 990.154,A -85,B 0,C 180,E1 10144.559,E2 10144.559} C_VEL
LIN {X 0,Y 396.85,Z 975.34,A -85,B 0,C 180,E1 10153.905,E2 10153.905} C_VEL
LIN {X 0,Y 401.938,Z 945.757,A -85,B 0,C 180,E1 10163.497,E2 10163.497} C_VEL
LIN {X 0,Y 412.499,Z 901.337,A -85,B 0,C 180,E1 10172.109,E2 10172.109} C_VEL
LIN {X 0,Y 424.979,Z 847.547,A -85,B 0,C 180,E1 10178.601,E2 10178.601} C_VEL
LIN {X 0,Y 436.291,Z 785.604,A -85,B 0,C 180,E1 10183.155,E2 10183.155} C_VEL
LIN {X 0,Y 436.97,Z 769.751,A -85,B 0,C 180,E1 10184.162,E2 10184.162} C_VEL
LIN {X 0,Y 410.522,Z 717.494,A -85,B 0,C 180,E1 10190.901,E2 10190.901} C_VEL
LIN {X 0,Y 394.047,Z 691.44,A -85,B 0,C 180,E1 10195.139,E2 10195.139} C_VEL
LIN {X 0,Y 393.555,Z 691.44,A -85,B 0,C 180,E1 10206.706,E2 10206.706} C_VEL
LIN {X 0,Y 393.572,Z 691.44,A -85,B 0,C 180,E1 10217.54,E2 10217.54} C_VEL
LIN {X 0,Y 393.731,Z 691.44,A -85,B 0,C 180,E1 10228.623,E2 10228.623} C_VEL
LIN {X 0,Y 393.832,Z 691.44,A -85,B 0,C 180,E1 10238.504,E2 10238.504} C_VEL
LIN {X 0,Y 394.739,Z 691.44,A -85,B 0,C 180,E1 10248.631,E2 10248.631} C_VEL
LIN {X 0,Y 395.037,Z 691.44,A -85,B 0,C 180,E1 10258.946,E2 10258.946} C_VEL
LIN {X 0,Y 394.738,Z 691.44,A -85,B 0,C 180,E1 10269.934,E2 10269.934} C_VEL
LIN {X 0,Y 394.167,Z 691.44,A -85,B 0,C 180,E1 10281.421,E2 10281.421} C_VEL
LIN {X 0,Y 393.753,Z 692.581,A -85,B 0,C 180,E1 10292.493,E2 10292.493} C_VEL
LIN {X 0,Y 430.48,Z 752.289,A -85,B 0,C 180,E1 10300.746,E2 10300.746} C_VEL
LIN {X 0,Y 440.072,Z 777.483,A -85,B 0,C 180,E1 10303.26,E2 10303.26} C_VEL
LIN {X 0,Y 430.224,Z 842.526,A -85,B 0,C 180,E1 10306.794,E2 10306.794} C_VEL
LIN {X 0,Y 417.8,Z 901.685,A -85,B 0,C 180,E1 10312.36,E2 10312.36} C_VEL
LIN {X 0,Y 406.3,Z 950.881,A -85,B 0,C 180,E1 10319.718,E2 10319.718} C_VEL
LIN {X 0,Y 398.737,Z 989,A -85,B 0,C 180,E1 10328.717,E2 10328.717} C_VEL
LIN {X 0,Y 395.799,Z 1011.884,A -85,B 0,C 180,E1 10337.825,E2 10337.825} C_VEL
LIN {X 0,Y 395.291,Z 1016.356,A -85,B 0,C 180,E1 10340.636,E2 10340.636} C_VEL
LIN {X 0,Y 387.14,Z 1021.056,A -85,B 0,C 180,E1 10345.667,E2 10345.667} C_VEL
LIN {X 0,Y 387.177,Z 1021.652,A -85,B 0,C 180,E1 10353.37,E2 10353.37} C_VEL
LIN {X 0,Y 387.555,Z 1011.497,A -85,B 0,C 180,E1 10362.436,E2 10362.436} C_VEL
LIN {X 0,Y 391.456,Z 986.824,A -85,B 0,C 180,E1 10372.208,E2 10372.208} C_VEL
LIN {X 0,Y 400.121,Z 946.717,A -85,B 0,C 180,E1 10381.489,E2 10381.489} C_VEL
LIN {X 0,Y 412.326,Z 894.599,A -85,B 0,C 180,E1 10389.045,E2 10389.045} C_VEL
LIN {X 0,Y 425.393,Z 833.728,A -85,B 0,C 180,E1 10394.487,E2 10394.487} C_VEL
LIN {X 0,Y 433.474,Z 774.477,A -85,B 0,C 180,E1 10397.757,E2 10397.757} C_VEL
LIN {X 0,Y 409.274,Z 726.931,A -85,B 0,C 180,E1 10404.113,E2 10404.113} C_VEL
LIN {X 0,Y 388.759,Z 697.741,A -85,B 0,C 180,E1 10410.558,E2 10410.558} C_VEL
LIN {X 0,Y 385.731,Z 691.44,A -85,B 0,C 180,E1 10412.277,E2 10412.277} C_VEL
LIN {X 0,Y 386.275,Z 691.44,A -85,B 0,C 180,E1 10422.895,E2 10422.895} C_VEL
LIN {X 0,Y 387.064,Z 691.44,A -85,B 0,C 180,E1 10434.402,E2 10434.402} C_VEL
LIN {X 0,Y 387.136,Z 693.282,A -85,B 0,C 180,E1 10437.111,E2 10437.111} C_VEL
LIN {X 0,Y 405.267,Z 719.025,A -85,B 0,C 180,E1 10443.244,E2 10443.244} C_VEL
LIN {X 0,Y 427.054,Z 762.46,A -85,B 0,C 180,E1 10449.687,E2 10449.687} C_VEL
LIN {X 0,Y 431.741,Z 782.604,A -85,B 0,C 180,E1 10451.809,E2 10451.809} C_VEL
LIN {X 0,Y 420.138,Z 843.139,A -85,B 0,C 180,E1 10456.086,E2 10456.086} C_VEL
LIN {X 0,Y 406.674,Z 897.997,A -85,B 0,C 180,E1 10462.548,E2 10462.548} C_VEL
LIN {X 0,Y 395.833,Z 941.629,A -85,B 0,C 180,E1 10470.797,E2 10470.797} C_VEL
LIN {X 0,Y 389.194,Z 973.062,A -85,B 0,C 180,E1 10480.505,E2 10480.505} C_VEL
LIN {X 0,Y 386.977,Z 989.207,A -85,B 0,C 180,E1 10489.906,E2 10489.906} C_VEL
LIN {X 0,Y 386.172,Z 993.54,A -85,B 0,C 180,E1 10497.96,E2 10497.96} C_VEL
LIN {X 0,Y 387.278,Z 987.95,A -85,B 0,C 180,E1 10507.087,E2 10507.087} C_VEL
LIN {X 0,Y 389.471,Z 970.046,A -85,B 0,C 180,E1 10516.556,E2 10516.556} C_VEL
LIN {X 0,Y 396.174,Z 938.434,A -85,B 0,C 180,E1 10525.848,E2 10525.848} C_VEL
LIN {X 0,Y 407.719,Z 893.149,A -85,B 0,C 180,E1 10534.003,E2 10534.003} C_VEL
LIN {X 0,Y 420.678,Z 838.922,A -85,B 0,C 180,E1 10540.13,E2 10540.13} C_VEL
LIN {X 0,Y 431.39,Z 774.311,A -85,B 0,C 180,E1 10544.626,E2 10544.626} C_VEL
LIN {X 0,Y 406.125,Z 722.967,A -85,B 0,C 180,E1 10551.447,E2 10551.447} C_VEL
LIN {X 0,Y 385.923,Z 691.44,A -85,B 0,C 180,E1 10556.888,E2 10556.888} C_VEL
LIN {X 0,Y 385.54,Z 691.44,A -85,B 0,C 180,E1 10567.6,E2 10567.6} C_VEL
LIN {X 0,Y 385.55,Z 691.44,A -85,B 0,C 180,E1 10576.737,E2 10576.737} C_VEL
LIN {X 0,Y 385.617,Z 691.44,A -85,B 0,C 180,E1 10587.885,E2 10587.885} C_VEL
LIN {X 0,Y 385.766,Z 691.44,A -85,B 0,C 180,E1 10598.032,E2 10598.032} C_VEL
LIN {X 0,Y 386.738,Z 691.44,A -85,B 0,C 180,E1 10607.513,E2 10607.513} C_VEL
LIN {X 0,Y 387.051,Z 691.44,A -85,B 0,C 180,E1 10619.008,E2 10619.008} C_VEL
LIN {X 0,Y 386.716,Z 691.44,A -85,B 0,C 180,E1 10630.142,E2 10630.142} C_VEL
LIN {X 0,Y 386.086,Z 691.44,A -85,B 0,C 180,E1 10641.893,E2 10641.893} C_VEL
LIN {X 0,Y 385.782,Z 692.8,A -85,B 0,C 180,E1 10650.812,E2 10650.812} C_VEL
LIN {X 0,Y 421.657,Z 749.9,A -85,B 0,C 180,E1 10659.337,E2 10659.337} C_VEL
LIN {X 0,Y 434.098,Z 779.986,A -85,B 0,C 180,E1 10662.606,E2 10662.606} C_VEL
LIN {X 0,Y 423.683,Z 844.606,A -85,B 0,C 180,E1 10666.23,E2 10666.23} C_VEL
LIN {X 0,Y 410.615,Z 903.804,A -85,B 0,C 180,E1 10671.949,E2 10671.949} C_VEL
LIN {X 0,Y 398.445,Z 953.514,A -85,B 0,C 180,E1 10679.69,E2 10679.69} C_VEL
LIN {X 0,Y 390.934,Z 988.936,A -85,B 0,C 180,E1 10688.358,E2 10688.358} C_VEL
LIN {X 0,Y 387.781,Z 1012.595,A -85,B 0,C 180,E1 10698.156,E2 10698.156} C_VEL
LIN {X 0,Y 387.14,Z 1021.056,A -85,B 0,C 180,E1 10705.667,E2 10705.667} C_VEL
LIN {X 0,Y 379.254,Z 1022.071,A -85,B 0,C 180,E1 10710.849,E2 10710.849} C_VEL
LIN {X 0,Y 379.3,Z 1014.829,A -85,B 0,C 180,E1 10720.371,E2 10720.371} C_VEL
LIN {X 0,Y 381.484,Z 996.932,A -85,B 0,C 180,E1 10729.158,E2 10729.158} C_VEL
LIN {X 0,Y 388.281,Z 964.176,A -85,B 0,C 180,E1 10738.509,E2 10738.509} C_VEL
LIN {X 0,Y 400.346,Z 916.024,A -85,B 0,C 180,E1 10747.017,E2 10747.017} C_VEL
LIN {X 0,Y 414.034,Z 859.705,A -85,B 0,C 180,E1 10753.232,E2 10753.232} C_VEL
LIN {X 0,Y 426.177,Z 797.098,A -85,B 0,C 180,E1 10757.382,E2 10757.382} C_VEL
LIN {X 0,Y 427.629,Z 777.844,A -85,B 0,C 180,E1 10758.415,E2 10758.415} C_VEL
LIN {X 0,Y 404.519,Z 730.852,A -85,B 0,C 180,E1 10764.974,E2 10764.974} C_VEL
LIN {X 0,Y 385.279,Z 703.666,A -85,B 0,C 180,E1 10771.448,E2 10771.448} C_VEL
LIN {X 0,Y 377.927,Z 691.44,A -85,B 0,C 180,E1 10775.73,E2 10775.73} C_VEL
LIN {X 0,Y 378.501,Z 691.44,A -85,B 0,C 180,E1 10787.291,E2 10787.291} C_VEL
LIN {X 0,Y 379.251,Z 693.474,A -85,B 0,C 180,E1 10793.927,E2 10793.927} C_VEL
LIN {X 0,Y 395.35,Z 715.324,A -85,B 0,C 180,E1 10800.662,E2 10800.662} C_VEL
LIN {X 0,Y 416.602,Z 754.283,A -85,B 0,C 180,E1 10807.43,E2 10807.43} C_VEL
LIN {X 0,Y 425.835,Z 785.407,A -85,B 0,C 180,E1 10811.163,E2 10811.163} C_VEL
LIN {X 0,Y 413.609,Z 845.595,A -85,B 0,C 180,E1 10815.536,E2 10815.536} C_VEL
LIN {X 0,Y 399.11,Z 901.582,A -85,B 0,C 180,E1 10822.359,E2 10822.359} C_VEL
LIN {X 0,Y 387.461,Z 945.572,A -85,B 0,C 180,E1 10831.135,E2 10831.135} C_VEL
LIN {X 0,Y 380.927,Z 975.563,A -85,B 0,C 180,E1 10841.121,E2 10841.121} C_VEL
LIN {X 0,Y 378.944,Z 989.975,A -85,B 0,C 180,E1 10850.207,E2 10850.207} C_VEL
LIN {X 0,Y 378.209,Z 993.569,A -85,B 0,C 180,E1 10859.897,E2 10859.897} C_VEL
LIN {X 0,Y 379.406,Z 986.112,A -85,B 0,C 180,E1 10868.894,E2 10868.894} C_VEL
LIN {X 0,Y 382.679,Z 966.008,A -85,B 0,C 180,E1 10878.564,E2 10878.564} C_VEL
LIN {X 0,Y 391.291,Z 929.93,A -85,B 0,C 180,E1 10888.334,E2 10888.334} C_VEL
LIN {X 0,Y 404.317,Z 881.297,A -85,B 0,C 180,E1 10896.327,E2 10896.327} C_VEL
LIN {X 0,Y 417.723,Z 824.916,A -85,B 0,C 180,E1 10902.059,E2 10902.059} C_VEL
LIN {X 0,Y 424.958,Z 776.622,A -85,B 0,C 180,E1 10905.365,E2 10905.365} C_VEL
LIN {X 0,Y 400.785,Z 727.258,A -85,B 0,C 180,E1 10912.221,E2 10912.221} C_VEL
LIN {X 0,Y 377.797,Z 691.44,A -85,B 0,C 180,E1 10918.815,E2 10918.815} C_VEL
LIN {X 0,Y 377.492,Z 691.44,A -85,B 0,C 180,E1 10928.546,E2 10928.546} C_VEL
LIN {X 0,Y 377.417,Z 691.44,A -85,B 0,C 180,E1 10938.412,E2 10938.412} C_VEL
LIN {X 0,Y 377.641,Z 691.44,A -85,B 0,C 180,E1 10949.823,E2 10949.823} C_VEL
LIN {X 0,Y 377.981,Z 691.44,A -85,B 0,C 180,E1 10960.655,E2 10960.655} C_VEL
LIN {X 0,Y 378.688,Z 691.44,A -85,B 0,C 180,E1 10969.586,E2 10969.586} C_VEL
LIN {X 0,Y 379.486,Z 691.44,A -85,B 0,C 180,E1 10981.119,E2 10981.119} C_VEL
LIN {X 0,Y 378.521,Z 691.44,A -85,B 0,C 180,E1 10992.709,E2 10992.709} C_VEL
LIN {X 0,Y 378.064,Z 691.44,A -85,B 0,C 180,E1 11002.382,E2 11002.382} C_VEL
LIN {X 0,Y 377.956,Z 693.315,A -85,B 0,C 180,E1 11009.059,E2 11009.059} C_VEL
LIN {X 0,Y 412.994,Z 747.937,A -85,B 0,C 180,E1 11017.879,E2 11017.879} C_VEL
LIN {X 0,Y 428.07,Z 783.023,A -85,B 0,C 180,E1 11021.952,E2 11021.952} C_VEL
LIN {X 0,Y 416.654,Z 849.219,A -85,B 0,C 180,E1 11025.844,E2 11025.844} C_VEL
LIN {X 0,Y 402.963,Z 907.483,A -85,B 0,C 180,E1 11031.752,E2 11031.752} C_VEL
LIN {X 0,Y 390.507,Z 956.099,A -85,B 0,C 180,E1 11039.654,E2 11039.654} C_VEL
LIN {X 0,Y 382.522,Z 993.186,A -85,B 0,C 180,E1 11049.419,E2 11049.419} C_VEL
LIN {X 0,Y 379.519,Z 1014.912,A -85,B 0,C 180,E1 11059.633,E2 11059.633} C_VEL
LIN {X 0,Y 378.963,Z 1022.065,A -85,B 0,C 180,E1 11068.852,E2 11068.852} C_VEL
LIN {X 0,Y 379.254,Z 1022.071,A -85,B 0,C 180,E1 11070.849,E2 11070.849} C_VEL
LIN {X 0,Y 371.212,Z 1019.401,A -85,B 0,C 180,E1 11076.118,E2 11076.118} C_VEL
LIN {X 0,Y 372.864,Z 1004.568,A -85,B 0,C 180,E1 11086.259,E2 11086.259} C_VEL
LIN {X 0,Y 378.508,Z 974.05,A -85,B 0,C 180,E1 11096.582,E2 11096.582} C_VEL
LIN {X 0,Y 389.521,Z 931.175,A -85,B 0,C 180,E1 11105.375,E2 11105.375} C_VEL
LIN {X 0,Y 403.82,Z 877.211,A -85,B 0,C 180,E1 11112.347,E2 11112.347} C_VEL
LIN {X 0,Y 417.728,Z 812.919,A -85,B 0,C 180,E1 11117.363,E2 11117.363} C_VEL
LIN {X 0,Y 421.877,Z 781.129,A -85,B 0,C 180,E1 11119.096,E2 11119.096} C_VEL
LIN {X 0,Y 400.458,Z 736.324,A -85,B 0,C 180,E1 11125.658,E2 11125.658} C_VEL
LIN {X 0,Y 380.608,Z 706.347,A -85,B 0,C 180,E1 11133.078,E2 11133.078} C_VEL
LIN {X 0,Y 372.896,Z 697.62,A -85,B 0,C 180,E1 11137.877,E2 11137.877} C_VEL
LIN {X 0,Y 370.179,Z 691.44,A -85,B 0,C 180,E1 11142.126,E2 11142.126} C_VEL
LIN {X 0,Y 370.819,Z 693.748,A -85,B 0,C 180,E1 11148.148,E2 11148.148} C_VEL
LIN {X 0,Y 378.005,Z 702.353,A -85,B 0,C 180,E1 11153.95,E2 11153.95} C_VEL
LIN {X 0,Y 393.448,Z 723.74,A -85,B 0,C 180,E1 11160.563,E2 11160.563} C_VEL
LIN {X 0,Y 412.891,Z 762.179,A -85,B 0,C 180,E1 11167.286,E2 11167.286} C_VEL
LIN {X 0,Y 420.043,Z 787.72,A -85,B 0,C 180,E1 11170.464,E2 11170.464} C_VEL
LIN {X 0,Y 407.343,Z 847.048,A -85,B 0,C 180,E1 11174.875,E2 11174.875} C_VEL
LIN {X 0,Y 392.289,Z 902.394,A -85,B 0,C 180,E1 11181.738,E2 11181.738} C_VEL
LIN {X 0,Y 380.465,Z 944.904,A -85,B 0,C 180,E1 11190.342,E2 11190.342} C_VEL
LIN {X 0,Y 373.264,Z 975.284,A -85,B 0,C 180,E1 11200.495,E2 11200.495} C_VEL
LIN {X 0,Y 371.133,Z 989.406,A -85,B 0,C 180,E1 11209.18,E2 11209.18} C_VEL
LIN {X 0,Y 370.161,Z 993.97,A -85,B 0,C 180,E1 11219.172,E2 11219.172} C_VEL
LIN {X 0,Y 371.399,Z 987.295,A -85,B 0,C 180,E1 11228.424,E2 11228.424} C_VEL
LIN {X 0,Y 374.56,Z 968.14,A -85,B 0,C 180,E1 11238.313,E2 11238.313} C_VEL
LIN {X 0,Y 382.876,Z 934.391,A -85,B 0,C 180,E1 11248.014,E2 11248.014} C_VEL
LIN {X 0,Y 395.899,Z 888.219,A -85,B 0,C 180,E1 11256.155,E2 11256.155} C_VEL
LIN {X 0,Y 410.294,Z 831.939,A -85,B 0,C 180,E1 11262.281,E2 11262.281} C_VEL
LIN {X 0,Y 418.856,Z 779.948,A -85,B 0,C 180,E1 11265.994,E2 11265.994} C_VEL
LIN {X 0,Y 395.356,Z 730.955,A -85,B 0,C 180,E1 11273.066,E2 11273.066} C_VEL
LIN {X 0,Y 369.618,Z 691.44,A -85,B 0,C 180,E1 11280.88,E2 11280.88} C_VEL
LIN {X 0,Y 369.36,Z 691.44,A -85,B 0,C 180,E1 11292.684,E2 11292.684} C_VEL
LIN {X 0,Y 369.353,Z 691.44,A -85,B 0,C 180,E1 11303.409,E2 11303.409} C_VEL
LIN {X 0,Y 369.651,Z 691.44,A -85,B 0,C 180,E1 11314.441,E2 11314.441} C_VEL
LIN {X 0,Y 370.647,Z 691.44,A -85,B 0,C 180,E1 11326.961,E2 11326.961} C_VEL
LIN {X 0,Y 371.061,Z 691.44,A -85,B 0,C 180,E1 11338.994,E2 11338.994} C_VEL
LIN {X 0,Y 370.649,Z 691.44,A -85,B 0,C 180,E1 11350.587,E2 11350.587} C_VEL
LIN {X 0,Y 370.015,Z 691.44,A -85,B 0,C 180,E1 11362.655,E2 11362.655} C_VEL
LIN {X 0,Y 370.019,Z 693.25,A -85,B 0,C 180,E1 11367.109,E2 11367.109} C_VEL
LIN {X 0,Y 405.064,Z 747.098,A -85,B 0,C 180,E1 11376.504,E2 11376.504} C_VEL
LIN {X 0,Y 422.103,Z 785.579,A -85,B 0,C 180,E1 11381.266,E2 11381.266} C_VEL
LIN {X 0,Y 410.01,Z 852.035,A -85,B 0,C 180,E1 11385.31,E2 11385.31} C_VEL
LIN {X 0,Y 395.733,Z 909.683,A -85,B 0,C 180,E1 11391.359,E2 11391.359} C_VEL
LIN {X 0,Y 382.838,Z 957.346,A -85,B 0,C 180,E1 11399.371,E2 11399.371} C_VEL
LIN {X 0,Y 374.685,Z 993.101,A -85,B 0,C 180,E1 11409.051,E2 11409.051} C_VEL
LIN {X 0,Y 371.573,Z 1014.612,A -85,B 0,C 180,E1 11419.408,E2 11419.408} C_VEL
LIN {X 0,Y 370.988,Z 1021.766,A -85,B 0,C 180,E1 11428.827,E2 11428.827} C_VEL
LIN {X 0,Y 371.212,Z 1019.401,A -85,B 0,C 180,E1 11436.118,E2 11436.118} C_VEL
LIN {X 0,Y 363.405,Z 1013.321,A -85,B 0,C 180,E1 11441.463,E2 11441.463} C_VEL
LIN {X 0,Y 366.576,Z 993.351,A -85,B 0,C 180,E1 11451.107,E2 11451.107} C_VEL
LIN {X 0,Y 375.31,Z 957.733,A -85,B 0,C 180,E1 11460.975,E2 11460.975} C_VEL
LIN {X 0,Y 388.758,Z 909.456,A -85,B 0,C 180,E1 11469.3,E2 11469.3} C_VEL
LIN {X 0,Y 404.115,Z 851.256,A -85,B 0,C 180,E1 11475.499,E2 11475.499} C_VEL
LIN {X 0,Y 416.39,Z 785.172,A -85,B 0,C 180,E1 11479.692,E2 11479.692} C_VEL
LIN {X 0,Y 396.231,Z 741.576,A -85,B 0,C 180,E1 11486.36,E2 11486.36} C_VEL
LIN {X 0,Y 378.142,Z 713.554,A -85,B 0,C 180,E1 11493.679,E2 11493.679} C_VEL
LIN {X 0,Y 370.67,Z 704.549,A -85,B 0,C 180,E1 11498.863,E2 11498.863} C_VEL
LIN {X 0,Y 368.912,Z 699.307,A -85,B 0,C 180,E1 11502.063,E2 11502.063} C_VEL
LIN {X 0,Y 369.597,Z 701.78,A -85,B 0,C 180,E1 11508.065,E2 11508.065} C_VEL
LIN {X 0,Y 376.736,Z 710.76,A -85,B 0,C 180,E1 11513.929,E2 11513.929} C_VEL
LIN {X 0,Y 391.727,Z 732.69,A -85,B 0,C 180,E1 11520.655,E2 11520.655} C_VEL
LIN {X 0,Y 409.832,Z 771.983,A -85,B 0,C 180,E1 11527.47,E2 11527.47} C_VEL
LIN {X 0,Y 413.919,Z 792.557,A -85,B 0,C 180,E1 11529.89,E2 11529.89} C_VEL
LIN {X 0,Y 399.942,Z 852.943,A -85,B 0,C 180,E1 11534.628,E2 11534.628} C_VEL
LIN {X 0,Y 384.792,Z 905.545,A -85,B 0,C 180,E1 11541.494,E2 11541.494} C_VEL
LIN {X 0,Y 372.541,Z 947.275,A -85,B 0,C 180,E1 11550.279,E2 11550.279} C_VEL
LIN {X 0,Y 365.548,Z 975.51,A -85,B 0,C 180,E1 11560.077,E2 11560.077} C_VEL
LIN {X 0,Y 363.073,Z 990.328,A -85,B 0,C 180,E1 11569.62,E2 11569.62} C_VEL
LIN {X 0,Y 362.188,Z 994.259,A -85,B 0,C 180,E1 11579.231,E2 11579.231} C_VEL
LIN {X 0,Y 363.368,Z 988.508,A -85,B 0,C 180,E1 11587.922,E2 11587.922} C_VEL
LIN {X 0,Y 366.214,Z 971.079,A -85,B 0,C 180,E1 11597.677,E2 11597.677} C_VEL
LIN {X 0,Y 374.46,Z 938.847,A -85,B 0,C 180,E1 11607.678,E2 11607.678} C_VEL
LIN {X 0,Y 388.048,Z 893.164,A -85,B 0,C 180,E1 11616.21,E2 11616.21} C_VEL
LIN {X 0,Y 402.86,Z 838.437,A -85,B 0,C 180,E1 11622.511,E2 11622.511} C_VEL
LIN {X 0,Y 413.178,Z 784.346,A -85,B 0,C 180,E1 11626.492,E2 11626.492} C_VEL
LIN {X 0,Y 390.762,Z 735.954,A -85,B 0,C 180,E1 11633.706,E2 11633.706} C_VEL
LIN {X 0,Y 363.74,Z 696.936,A -85,B 0,C 180,E1 11641.738,E2 11641.738} C_VEL
LIN {X 0,Y 361.588,Z 691.44,A -85,B 0,C 180,E1 11642.662,E2 11642.662} C_VEL
LIN {X 0,Y 361.352,Z 691.44,A -85,B 0,C 180,E1 11653.866,E2 11653.866} C_VEL
LIN {X 0,Y 361.339,Z 691.44,A -85,B 0,C 180,E1 11665.436,E2 11665.436} C_VEL
LIN {X 0,Y 361.629,Z 691.44,A -85,B 0,C 180,E1 11676.481,E2 11676.481} C_VEL
LIN {X 0,Y 362.59,Z 691.44,A -85,B 0,C 180,E1 11686.666,E2 11686.666} C_VEL
LIN {X 0,Y 363.043,Z 691.44,A -85,B 0,C 180,E1 11698.775,E2 11698.775} C_VEL
LIN {X 0,Y 362.643,Z 691.44,A -85,B 0,C 180,E1 11710.438,E2 11710.438} C_VEL
LIN {X 0,Y 362.036,Z 691.44,A -85,B 0,C 180,E1 11720.838,E2 11720.838} C_VEL
LIN {X 0,Y 361.959,Z 692.823,A -85,B 0,C 180,E1 11724.938,E2 11724.938} C_VEL
LIN {X 0,Y 395.482,Z 743.699,A -85,B 0,C 180,E1 11734.617,E2 11734.617} C_VEL
LIN {X 0,Y 416.201,Z 787.92,A -85,B 0,C 180,E1 11740.569,E2 11740.569} C_VEL
LIN {X 0,Y 403.552,Z 854.018,A -85,B 0,C 180,E1 11744.694,E2 11744.694} C_VEL
LIN {X 0,Y 388.247,Z 912.864,A -85,B 0,C 180,E1 11751.083,E2 11751.083} C_VEL
LIN {X 0,Y 374.675,Z 960.812,A -85,B 0,C 180,E1 11759.581,E2 11759.581} C_VEL
LIN {X 0,Y 366.585,Z 994.933,A -85,B 0,C 180,E1 11769.396,E2 11769.396} C_VEL
LIN {X 0,Y 363.618,Z 1014.311,A -85,B 0,C 180,E1 11779.174,E2 11779.174} C_VEL
LIN {X 0,Y 362.992,Z 1021.469,A -85,B 0,C 180,E1 11788.801,E2 11788.801} C_VEL
LIN {X 0,Y 363.383,Z 1017.114,A -85,B 0,C 180,E1 11798.404,E2 11798.404} C_VEL
LIN {X 0,Y 363.405,Z 1013.321,A -85,B 0,C 180,E1 11801.463,E2 11801.463} C_VEL
LIN {X 0,Y 356.991,Z 1004.159,A -85,B 0,C 180,E1 11806.848,E2 11806.848} C_VEL
LIN {X 0,Y 363.132,Z 974.736,A -85,B 0,C 180,E1 11817.367,E2 11817.367} C_VEL
LIN {X 0,Y 375.522,Z 931.982,A -85,B 0,C 180,E1 11826.589,E2 11826.589} C_VEL
LIN {X 0,Y 391.448,Z 877.707,A -85,B 0,C 180,E1 11833.853,E2 11833.853} C_VEL
LIN {X 0,Y 406.688,Z 813.519,A -85,B 0,C 180,E1 11838.987,E2 11838.987} C_VEL
LIN {X 0,Y 410.529,Z 788.15,A -85,B 0,C 180,E1 11840.442,E2 11840.442} C_VEL
LIN {X 0,Y 391.393,Z 745.253,A -85,B 0,C 180,E1 11847.361,E2 11847.361} C_VEL
LIN {X 0,Y 375.161,Z 720.118,A -85,B 0,C 180,E1 11854.582,E2 11854.582} C_VEL
LIN {X 0,Y 368.786,Z 711.55,A -85,B 0,C 180,E1 11859.714,E2 11859.714} C_VEL
LIN {X 0,Y 367.311,Z 707.134,A -85,B 0,C 180,E1 11864.454,E2 11864.454} C_VEL
LIN {X 0,Y 373.429,Z 715.196,A -85,B 0,C 180,E1 11872.594,E2 11872.594} C_VEL
LIN {X 0,Y 388.707,Z 739.839,A -85,B 0,C 180,E1 11880.301,E2 11880.301} C_VEL
LIN {X 0,Y 405.655,Z 779.375,A -85,B 0,C 180,E1 11887.287,E2 11887.287} C_VEL
LIN {X 0,Y 408.221,Z 794.985,A -85,B 0,C 180,E1 11889.168,E2 11889.168} C_VEL
LIN {X 0,Y 393.354,Z 855.981,A -85,B 0,C 180,E1 11894.085,E2 11894.085} C_VEL
LIN {X 0,Y 377.148,Z 909.127,A -85,B 0,C 180,E1 11901.306,E2 11901.306} C_VEL
LIN {X 0,Y 364.172,Z 950.776,A -85,B 0,C 180,E1 11910.583,E2 11910.583} C_VEL
LIN {X 0,Y 356.985,Z 979.05,A -85,B 0,C 180,E1 11921.243,E2 11921.243} C_VEL
LIN {X 0,Y 355.069,Z 990.861,A -85,B 0,C 180,E1 11929.67,E2 11929.67} C_VEL
LIN {X 0,Y 354.234,Z 994.363,A -85,B 0,C 180,E1 11940.485,E2 11940.485} C_VEL
LIN {X 0,Y 355.847,Z 985.814,A -85,B 0,C 180,E1 11950.469,E2 11950.469} C_VEL
LIN {X 0,Y 360.906,Z 963.074,A -85,B 0,C 180,E1 11961.267,E2 11961.267} C_VEL
LIN {X 0,Y 371.121,Z 927.523,A -85,B 0,C 180,E1 11970.88,E2 11970.88} C_VEL
LIN {X 0,Y 385.796,Z 879.316,A -85,B 0,C 180,E1 11978.911,E2 11978.911} C_VEL
LIN {X 0,Y 401.46,Z 820.015,A -85,B 0,C 180,E1 11984.868,E2 11984.868} C_VEL
LIN {X 0,Y 407.232,Z 787.858,A -85,B 0,C 180,E1 11987.12,E2 11987.12} C_VEL
LIN {X 0,Y 386.022,Z 741.142,A -85,B 0,C 180,E1 11994.341,E2 11994.341} C_VEL
LIN {X 0,Y 359.754,Z 702.175,A -85,B 0,C 180,E1 12002.613,E2 12002.613} C_VEL
LIN {X 0,Y 353.338,Z 691.44,A -85,B 0,C 180,E1 12005.44,E2 12005.44} C_VEL
LIN {X 0,Y 353.288,Z 691.44,A -85,B 0,C 180,E1 12015.137,E2 12015.137} C_VEL
LIN {X 0,Y 353.357,Z 691.44,A -85,B 0,C 180,E1 12027.506,E2 12027.506} C_VEL
LIN {X 0,Y 353.672,Z 691.44,A -85,B 0,C 180,E1 12038.584,E2 12038.584} C_VEL
LIN {X 0,Y 354.636,Z 691.44,A -85,B 0,C 180,E1 12048.871,E2 12048.871} C_VEL
LIN {X 0,Y 355.457,Z 691.44,A -85,B 0,C 180,E1 12061.195,E2 12061.195} C_VEL
LIN {X 0,Y 354.374,Z 691.44,A -85,B 0,C 180,E1 12073.591,E2 12073.591} C_VEL
LIN {X 0,Y 354.049,Z 693.182,A -85,B 0,C 180,E1 12082.636,E2 12082.636} C_VEL
LIN {X 0,Y 384.711,Z 738.275,A -85,B 0,C 180,E1 12092.221,E2 12092.221} C_VEL
LIN {X 0,Y 409.699,Z 787.653,A -85,B 0,C 180,E1 12099.566,E2 12099.566} C_VEL
LIN {X 0,Y 397.808,Z 853.301,A -85,B 0,C 180,E1 12103.845,E2 12103.845} C_VEL
LIN {X 0,Y 382.334,Z 910.32,A -85,B 0,C 180,E1 12110.015,E2 12110.015} C_VEL
LIN {X 0,Y 368.357,Z 956.828,A -85,B 0,C 180,E1 12118.093,E2 12118.093} C_VEL
LIN {X 0,Y 358.994,Z 993.321,A -85,B 0,C 180,E1 12128.416,E2 12128.416} C_VEL
LIN {X 0,Y 355.659,Z 1014.01,A -85,B 0,C 180,E1 12138.928,E2 12138.928} C_VEL
LIN {X 0,Y 354.999,Z 1021.171,A -85,B 0,C 180,E1 12148.774,E2 12148.774} C_VEL
LIN {X 0,Y 355.372,Z 1016.798,A -85,B 0,C 180,E1 12158.595,E2 12158.595} C_VEL
LIN {X 0,Y 356.991,Z 1004.159,A -85,B 0,C 180,E1 12166.848,E2 12166.848} C_VEL
LIN {X 0,Y 351.314,Z 992.348,A -85,B 0,C 180,E1 12172.186,E2 12172.186} C_VEL
LIN {X 0,Y 361.392,Z 956.028,A -85,B 0,C 180,E1 12182.559,E2 12182.559} C_VEL
LIN {X 0,Y 376.497,Z 907.252,A -85,B 0,C 180,E1 12191.11,E2 12191.11} C_VEL
LIN {X 0,Y 393.075,Z 849.574,A -85,B 0,C 180,E1 12197.304,E2 12197.304} C_VEL
LIN {X 0,Y 404.808,Z 791.242,A -85,B 0,C 180,E1 12201.206,E2 12201.206} C_VEL
LIN {X 0,Y 387.157,Z 750.374,A -85,B 0,C 180,E1 12208.172,E2 12208.172} C_VEL
LIN {X 0,Y 372.824,Z 727.073,A -85,B 0,C 180,E1 12215.171,E2 12215.171} C_VEL
LIN {X 0,Y 366.442,Z 715.093,A -85,B 0,C 180,E1 12222.56,E2 12222.56} C_VEL
LIN {X 0,Y 367.193,Z 717.989,A -85,B 0,C 180,E1 12228.095,E2 12228.095} C_VEL
LIN {X 0,Y 373.894,Z 727.251,A -85,B 0,C 180,E1 12233.938,E2 12233.938} C_VEL
LIN {X 0,Y 386.89,Z 749.795,A -85,B 0,C 180,E1 12240.576,E2 12240.576} C_VEL
LIN {X 0,Y 401.74,Z 788.601,A -85,B 0,C 180,E1 12247.404,E2 12247.404} C_VEL
LIN {X 0,Y 401.988,Z 800.099,A -85,B 0,C 180,E1 12248.587,E2 12248.587} C_VEL
LIN {X 0,Y 386.959,Z 858.509,A -85,B 0,C 180,E1 12253.47,E2 12253.47} C_VEL
LIN {X 0,Y 369.806,Z 911.781,A -85,B 0,C 180,E1 12260.947,E2 12260.947} C_VEL
LIN {X 0,Y 356.417,Z 952.45,A -85,B 0,C 180,E1 12270.371,E2 12270.371} C_VEL
LIN {X 0,Y 349.363,Z 978.732,A -85,B 0,C 180,E1 12280.522,E2 12280.522} C_VEL
LIN {X 0,Y 346.835,Z 992.2,A -85,B 0,C 180,E1 12290.622,E2 12290.622} C_VEL
LIN {X 0,Y 346.114,Z 994.8,A -85,B 0,C 180,E1 12299.721,E2 12299.721} C_VEL
LIN {X 0,Y 347.684,Z 987.314,A -85,B 0,C 180,E1 12309.837,E2 12309.837} C_VEL
LIN {X 0,Y 352.401,Z 966.275,A -85,B 0,C 180,E1 12320.708,E2 12320.708} C_VEL
LIN {X 0,Y 363.141,Z 930.93,A -85,B 0,C 180,E1 12330.899,E2 12330.899} C_VEL
LIN {X 0,Y 378.478,Z 882.99,A -85,B 0,C 180,E1 12339.231,E2 12339.231} C_VEL
LIN {X 0,Y 394.315,Z 826.388,A -85,B 0,C 180,E1 12345.205,E2 12345.205} C_VEL
LIN {X 0,Y 401.232,Z 791.227,A -85,B 0,C 180,E1 12347.794,E2 12347.794} C_VEL
LIN {X 0,Y 381.141,Z 746.017,A -85,B 0,C 180,E1 12355.045,E2 12355.045} C_VEL
LIN {X 0,Y 354.742,Z 705.455,A -85,B 0,C 180,E1 12363.921,E2 12363.921} C_VEL
LIN {X 0,Y 345.301,Z 691.44,A -85,B 0,C 180,E1 12368.289,E2 12368.289} C_VEL
LIN {X 0,Y 345.181,Z 691.44,A -85,B 0,C 180,E1 12380.369,E2 12380.369} C_VEL
LIN {X 0,Y 345.485,Z 691.44,A -85,B 0,C 180,E1 12392.508,E2 12392.508} C_VEL
LIN {X 0,Y 346.196,Z 691.44,A -85,B 0,C 180,E1 12403.419,E2 12403.419} C_VEL
LIN {X 0,Y 346.818,Z 691.44,A -85,B 0,C 180,E1 12413.692,E2 12413.692} C_VEL
LIN {X 0,Y 346.942,Z 691.44,A -85,B 0,C 180,E1 12423.732,E2 12423.732} C_VEL
LIN {X 0,Y 346.351,Z 691.44,A -85,B 0,C 180,E1 12433.912,E2 12433.912} C_VEL
LIN {X 0,Y 346.085,Z 692.916,A -85,B 0,C 180,E1 12440.041,E2 12440.041} C_VEL
LIN {X 0,Y 376.037,Z 736.379,A -85,B 0,C 180,E1 12450.257,E2 12450.257} C_VEL
LIN {X 0,Y 400.962,Z 783.898,A -85,B 0,C 180,E1 12457.894,E2 12457.894} C_VEL
LIN {X 0,Y 403.964,Z 796.671,A -85,B 0,C 180,E1 12459.315,E2 12459.315} C_VEL
LIN {X 0,Y 389.594,Z 861.659,A -85,B 0,C 180,E1 12463.75,E2 12463.75} C_VEL
LIN {X 0,Y 373.471,Z 917.998,A -85,B 0,C 180,E1 12470.384,E2 12470.384} C_VEL
LIN {X 0,Y 358.984,Z 964.632,A -85,B 0,C 180,E1 12479.325,E2 12479.325} C_VEL
LIN {X 0,Y 350.5,Z 997.442,A -85,B 0,C 180,E1 12489.733,E2 12489.733} C_VEL
LIN {X 0,Y 347.43,Z 1015.463,A -85,B 0,C 180,E1 12500.062,E2 12500.062} C_VEL
LIN {X 0,Y 347.003,Z 1020.873,A -85,B 0,C 180,E1 12508.746,E2 12508.746} C_VEL
LIN {X 0,Y 347.357,Z 1016.481,A -85,B 0,C 180,E1 12518.795,E2 12518.795} C_VEL
LIN {X 0,Y 349.485,Z 1000.063,A -85,B 0,C 180,E1 12529.005,E2 12529.005} C_VEL
LIN {X 0,Y 351.314,Z 992.348,A -85,B 0,C 180,E1 12532.186,E2 12532.186} C_VEL
LIN {X 0,Y 347.312,Z 977.935,A -85,B 0,C 180,E1 12537.492,E2 12537.492} C_VEL
LIN {X 0,Y 361.057,Z 934.817,A -85,B 0,C 180,E1 12547.549,E2 12547.549} C_VEL
LIN {X 0,Y 378.334,Z 881.536,A -85,B 0,C 180,E1 12555.1,E2 12555.1} C_VEL
LIN {X 0,Y 394.955,Z 819.159,A -85,B 0,C 180,E1 12560.407,E2 12560.407} C_VEL
LIN {X 0,Y 399.091,Z 794.298,A -85,B 0,C 180,E1 12562.015,E2 12562.015} C_VEL
LIN {X 0,Y 382.872,Z 755.403,A -85,B 0,C 180,E1 12568.986,E2 12568.986} C_VEL
LIN {X 0,Y 370.154,Z 733.484,A -85,B 0,C 180,E1 12575.993,E2 12575.993} C_VEL
LIN {X 0,Y 364.863,Z 722.931,A -85,B 0,C 180,E1 12584.347,E2 12584.347} C_VEL
LIN {X 0,Y 370.202,Z 732,A -85,B 0,C 180,E1 12592.521,E2 12592.521} C_VEL
LIN {X 0,Y 382.315,Z 753.99,A -85,B 0,C 180,E1 12599.6,E2 12599.6} C_VEL
LIN {X 0,Y 396.156,Z 791.781,A -85,B 0,C 180,E1 12606.623,E2 12606.623} C_VEL
LIN {X 0,Y 396.232,Z 803.593,A -85,B 0,C 180,E1 12607.887,E2 12607.887} C_VEL
LIN {X 0,Y 379.995,Z 862.79,A -85,B 0,C 180,E1 12613.049,E2 12613.049} C_VEL
LIN {X 0,Y 362.376,Z 914.772,A -85,B 0,C 180,E1 12620.649,E2 12620.649} C_VEL
LIN {X 0,Y 348.428,Z 954.831,A -85,B 0,C 180,E1 12630.361,E2 12630.361} C_VEL
LIN {X 0,Y 341.136,Z 980.716,A -85,B 0,C 180,E1 12641.061,E2 12641.061} C_VEL
LIN {X 0,Y 339.088,Z 991.715,A -85,B 0,C 180,E1 12649.539,E2 12649.539} C_VEL
LIN {X 0,Y 338.107,Z 995.213,A -85,B 0,C 180,E1 12658.925,E2 12658.925} C_VEL
LIN {X 0,Y 339.592,Z 988.524,A -85,B 0,C 180,E1 12669.335,E2 12669.335} C_VEL
LIN {X 0,Y 344.241,Z 968.486,A -85,B 0,C 180,E1 12680.485,E2 12680.485} C_VEL
LIN {X 0,Y 355.579,Z 932.786,A -85,B 0,C 180,E1 12691.224,E2 12691.224} C_VEL
LIN {X 0,Y 371.021,Z 886.842,A -85,B 0,C 180,E1 12699.53,E2 12699.53} C_VEL
LIN {X 0,Y 387.909,Z 829.775,A -85,B 0,C 180,E1 12705.8,E2 12705.8} C_VEL
LIN {X 0,Y 395.195,Z 794.646,A -85,B 0,C 180,E1 12708.455,E2 12708.455} C_VEL
LIN {X 0,Y 375.607,Z 749.242,A -85,B 0,C 180,E1 12716.032,E2 12716.032} C_VEL
LIN {X 0,Y 350.543,Z 711.134,A -85,B 0,C 180,E1 12724.904,E2 12724.904} C_VEL
LIN {X 0,Y 337.104,Z 691.44,A -85,B 0,C 180,E1 12730.752,E2 12730.752} C_VEL
LIN {X 0,Y 337.086,Z 691.44,A -85,B 0,C 180,E1 12742.544,E2 12742.544} C_VEL
LIN {X 0,Y 337.507,Z 691.44,A -85,B 0,C 180,E1 12754.686,E2 12754.686} C_VEL
LIN {X 0,Y 338.405,Z 691.44,A -85,B 0,C 180,E1 12765.694,E2 12765.694} C_VEL
LIN {X 0,Y 338.915,Z 691.44,A -85,B 0,C 180,E1 12776.12,E2 12776.12} C_VEL
LIN {X 0,Y 338.687,Z 691.44,A -85,B 0,C 180,E1 12786.4,E2 12786.4} C_VEL
LIN {X 0,Y 338.327,Z 693.401,A -85,B 0,C 180,E1 12797.252,E2 12797.252} C_VEL
LIN {X 0,Y 365.985,Z 732.307,A -85,B 0,C 180,E1 12807.684,E2 12807.684} C_VEL
LIN {X 0,Y 391.707,Z 779.503,A -85,B 0,C 180,E1 12815.996,E2 12815.996} C_VEL
LIN {X 0,Y 398.079,Z 799.464,A -85,B 0,C 180,E1 12818.598,E2 12818.598} C_VEL
LIN {X 0,Y 382.729,Z 865.463,A -85,B 0,C 180,E1 12823.264,E2 12823.264} C_VEL
LIN {X 0,Y 365.643,Z 921.94,A -85,B 0,C 180,E1 12830.239,E2 12830.239} C_VEL
LIN {X 0,Y 351.135,Z 966.363,A -85,B 0,C 180,E1 12839.183,E2 12839.183} C_VEL
LIN {X 0,Y 342.421,Z 998.664,A -85,B 0,C 180,E1 12849.91,E2 12849.91} C_VEL
LIN {X 0,Y 339.256,Z 1016.289,A -85,B 0,C 180,E1 12860.991,E2 12860.991} C_VEL
LIN {X 0,Y 339.347,Z 1020.568,A -85,B 0,C 180,E1 12871.28,E2 12871.28} C_VEL
LIN {X 0,Y 339.428,Z 1013.218,A -85,B 0,C 180,E1 12881.606,E2 12881.606} C_VEL
LIN {X 0,Y 343.413,Z 992.826,A -85,B 0,C 180,E1 12892.376,E2 12892.376} C_VEL
LIN {X 0,Y 347.312,Z 977.935,A -85,B 0,C 180,E1 12897.492,E2 12897.492} C_VEL
LIN {X 0,Y 345.35,Z 961.194,A -85,B 0,C 180,E1 12902.662,E2 12902.662} C_VEL
LIN {X 0,Y 361.605,Z 914.018,A -85,B 0,C 180,E1 12911.777,E2 12911.777} C_VEL
LIN {X 0,Y 379.732,Z 857.743,A -85,B 0,C 180,E1 12918.372,E2 12918.372} C_VEL
LIN {X 0,Y 393.686,Z 798.134,A -85,B 0,C 180,E1 12922.706,E2 12922.706} C_VEL
LIN {X 0,Y 378.518,Z 759.653,A -85,B 0,C 180,E1 12929.962,E2 12929.962} C_VEL
LIN {X 0,Y 366.454,Z 737.286,A -85,B 0,C 180,E1 12937.866,E2 12937.866} C_VEL
LIN {X 0,Y 363.494,Z 730.783,A -85,B 0,C 180,E1 12944.287,E2 12944.287} C_VEL
LIN {X 0,Y 368.85,Z 741.062,A -85,B 0,C 180,E1 12952.865,E2 12952.865} C_VEL
LIN {X 0,Y 379.799,Z 762.982,A -85,B 0,C 180,E1 12959.74,E2 12959.74} C_VEL
LIN {X 0,Y 391.836,Z 800.549,A -85,B 0,C 180,E1 12966.698,E2 12966.698} C_VEL
LIN {X 0,Y 375.088,Z 860.937,A -85,B 0,C 180,E1 12971.897,E2 12971.897} C_VEL
LIN {X 0,Y 356.161,Z 914.439,A -85,B 0,C 180,E1 12979.704,E2 12979.704} C_VEL
LIN {X 0,Y 341.084,Z 955.49,A -85,B 0,C 180,E1 12989.819,E2 12989.819} C_VEL
LIN {X 0,Y 333.099,Z 982.051,A -85,B 0,C 180,E1 13001.261,E2 13001.261} C_VEL
LIN {X 0,Y 330.561,Z 993.723,A -85,B 0,C 180,E1 13011.702,E2 13011.702} C_VEL
LIN {X 0,Y 330.225,Z 995.063,A -85,B 0,C 180,E1 13021.15,E2 13021.15} C_VEL
LIN {X 0,Y 332.167,Z 986.673,A -85,B 0,C 180,E1 13031.35,E2 13031.35} C_VEL
LIN {X 0,Y 338.341,Z 963.353,A -85,B 0,C 180,E1 13043.092,E2 13043.092} C_VEL
LIN {X 0,Y 351.01,Z 926.433,A -85,B 0,C 180,E1 13053.42,E2 13053.42} C_VEL
LIN {X 0,Y 367.806,Z 878.014,A -85,B 0,C 180,E1 13061.605,E2 13061.605} C_VEL
LIN {X 0,Y 384.954,Z 819.562,A -85,B 0,C 180,E1 13067.523,E2 13067.523} C_VEL
LIN {X 0,Y 388.669,Z 796.541,A -85,B 0,C 180,E1 13069.385,E2 13069.385} C_VEL
LIN {X 0,Y 370.167,Z 753.153,A -85,B 0,C 180,E1 13076.948,E2 13076.948} C_VEL
LIN {X 0,Y 346.402,Z 716.133,A -85,B 0,C 180,E1 13085.941,E2 13085.941} C_VEL
LIN {X 0,Y 329.091,Z 691.44,A -85,B 0,C 180,E1 13094.346,E2 13094.346} C_VEL
LIN {X 0,Y 329.08,Z 691.44,A -85,B 0,C 180,E1 13104.771,E2 13104.771} C_VEL
LIN {X 0,Y 329.515,Z 691.44,A -85,B 0,C 180,E1 13116.927,E2 13116.927} C_VEL
LIN {X 0,Y 330.5,Z 691.44,A -85,B 0,C 180,E1 13128.047,E2 13128.047} C_VEL
LIN {X 0,Y 331.049,Z 691.44,A -85,B 0,C 180,E1 13139.053,E2 13139.053} C_VEL
LIN {X 0,Y 330.616,Z 691.44,A -85,B 0,C 180,E1 13149.279,E2 13149.279} C_VEL
LIN {X 0,Y 330.482,Z 693.207,A -85,B 0,C 180,E1 13154,E2 13154} C_VEL
LIN {X 0,Y 355.798,Z 728.518,A -85,B 0,C 180,E1 13164.789,E2 13164.789} C_VEL
LIN {X 0,Y 381.543,Z 773.112,A -85,B 0,C 180,E1 13173.626,E2 13173.626} C_VEL
LIN {X 0,Y 392.281,Z 801.992,A -85,B 0,C 180,E1 13177.855,E2 13177.855} C_VEL
LIN {X 0,Y 376.948,Z 865.159,A -85,B 0,C 180,E1 13182.386,E2 13182.386} C_VEL
LIN {X 0,Y 359.196,Z 921.391,A -85,B 0,C 180,E1 13189.378,E2 13189.378} C_VEL
LIN {X 0,Y 343.975,Z 965.729,A -85,B 0,C 180,E1 13198.403,E2 13198.403} C_VEL
LIN {X 0,Y 334.564,Z 998.654,A -85,B 0,C 180,E1 13209.58,E2 13209.58} C_VEL
LIN {X 0,Y 331.288,Z 1015.986,A -85,B 0,C 180,E1 13220.773,E2 13220.773} C_VEL
LIN {X 0,Y 331.343,Z 1020.268,A -85,B 0,C 180,E1 13231.311,E2 13231.311} C_VEL
LIN {X 0,Y 331.482,Z 1012.9,A -85,B 0,C 180,E1 13241.888,E2 13241.888} C_VEL
LIN {X 0,Y 336.09,Z 991.615,A -85,B 0,C 180,E1 13253.271,E2 13253.271} C_VEL
LIN {X 0,Y 345.35,Z 961.194,A -85,B 0,C 180,E1 13262.662,E2 13262.662} C_VEL
LIN {X 0,Y 344.97,Z 942.247,A -85,B 0,C 180,E1 13267.663,E2 13267.663} C_VEL
LIN {X 0,Y 364.015,Z 889.465,A -85,B 0,C 180,E1 13275.984,E2 13275.984} C_VEL
LIN {X 0,Y 382.965,Z 826.727,A -85,B 0,C 180,E1 13281.789,E2 13281.789} C_VEL
LIN {X 0,Y 388.27,Z 801.764,A -85,B 0,C 180,E1 13283.453,E2 13283.453} C_VEL
LIN {X 0,Y 374.437,Z 764.953,A -85,B 0,C 180,E1 13290.804,E2 13290.804} C_VEL
LIN {X 0,Y 364.261,Z 744.701,A -85,B 0,C 180,E1 13298.335,E2 13298.335} C_VEL
LIN {X 0,Y 361.85,Z 738.596,A -85,B 0,C 180,E1 13304.213,E2 13304.213} C_VEL
LIN {X 0,Y 366.772,Z 749.161,A -85,B 0,C 180,E1 13312.891,E2 13312.891} C_VEL
LIN {X 0,Y 376.848,Z 771.472,A -85,B 0,C 180,E1 13319.76,E2 13319.76} C_VEL
LIN {X 0,Y 386.152,Z 805.554,A -85,B 0,C 180,E1 13326.088,E2 13326.088} C_VEL
LIN {X 0,Y 368.611,Z 864.12,A -85,B 0,C 180,E1 13331.293,E2 13331.293} C_VEL
LIN {X 0,Y 349.403,Z 915.708,A -85,B 0,C 180,E1 13339.037,E2 13339.037} C_VEL
LIN {X 0,Y 334.043,Z 955.395,A -85,B 0,C 180,E1 13349.013,E2 13349.013} C_VEL
LIN {X 0,Y 325.436,Z 981.914,A -85,B 0,C 180,E1 13360.561,E2 13360.561} C_VEL
LIN {X 0,Y 322.685,Z 993.655,A -85,B 0,C 180,E1 13370.928,E2 13370.928} C_VEL
LIN {X 0,Y 322.152,Z 995.571,A -85,B 0,C 180,E1 13380.672,E2 13380.672} C_VEL
LIN {X 0,Y 324.007,Z 987.981,A -85,B 0,C 180,E1 13390.862,E2 13390.862} C_VEL
LIN {X 0,Y 330.133,Z 966.01,A -85,B 0,C 180,E1 13402.727,E2 13402.727} C_VEL
LIN {X 0,Y 342.556,Z 931.188,A -85,B 0,C 180,E1 13413.185,E2 13413.185} C_VEL
LIN {X 0,Y 360.234,Z 882.797,A -85,B 0,C 180,E1 13421.853,E2 13421.853} C_VEL
LIN {X 0,Y 378.063,Z 825.282,A -85,B 0,C 180,E1 13427.975,E2 13427.975} C_VEL
LIN {X 0,Y 383.099,Z 801.142,A -85,B 0,C 180,E1 13429.9,E2 13429.9} C_VEL
LIN {X 0,Y 365.452,Z 758.211,A -85,B 0,C 180,E1 13437.635,E2 13437.635} C_VEL
LIN {X 0,Y 341.712,Z 719.956,A -85,B 0,C 180,E1 13447.284,E2 13447.284} C_VEL
LIN {X 0,Y 323.824,Z 697.498,A -85,B 0,C 180,E1 13456.142,E2 13456.142} C_VEL
LIN {X 0,Y 321.048,Z 691.44,A -85,B 0,C 180,E1 13458.33,E2 13458.33} C_VEL
LIN {X 0,Y 321.306,Z 691.44,A -85,B 0,C 180,E1 13470.905,E2 13470.905} C_VEL
LIN {X 0,Y 321.918,Z 691.44,A -85,B 0,C 180,E1 13482.128,E2 13482.128} C_VEL
LIN {X 0,Y 322.751,Z 691.44,A -85,B 0,C 180,E1 13493.219,E2 13493.219} C_VEL
LIN {X 0,Y 322.878,Z 691.44,A -85,B 0,C 180,E1 13504.011,E2 13504.011} C_VEL
LIN {X 0,Y 322.681,Z 693.186,A -85,B 0,C 180,E1 13510.209,E2 13510.209} C_VEL
LIN {X 0,Y 344.255,Z 722.877,A -85,B 0,C 180,E1 13520.952,E2 13520.952} C_VEL
LIN {X 0,Y 368.599,Z 761.99,A -85,B 0,C 180,E1 13530.078,E2 13530.078} C_VEL
LIN {X 0,Y 386.782,Z 802.758,A -85,B 0,C 180,E1 13536.98,E2 13536.98} C_VEL
LIN {X 0,Y 370.797,Z 866.315,A -85,B 0,C 180,E1 13541.625,E2 13541.625} C_VEL
LIN {X 0,Y 352.412,Z 922.179,A -85,B 0,C 180,E1 13548.703,E2 13548.703} C_VEL
LIN {X 0,Y 336.399,Z 966.555,A -85,B 0,C 180,E1 13557.988,E2 13557.988} C_VEL
LIN {X 0,Y 326.744,Z 998.403,A -85,B 0,C 180,E1 13569.116,E2 13569.116} C_VEL
LIN {X 0,Y 323.333,Z 1015.678,A -85,B 0,C 180,E1 13580.544,E2 13580.544} C_VEL
LIN {X 0,Y 323.352,Z 1019.966,A -85,B 0,C 180,E1 13591.343,E2 13591.343} C_VEL
LIN {X 0,Y 323.538,Z 1012.587,A -85,B 0,C 180,E1 13602.184,E2 13602.184} C_VEL
LIN {X 0,Y 328.538,Z 991.289,A -85,B 0,C 180,E1 13613.839,E2 13613.839} C_VEL
LIN {X 0,Y 340.958,Z 953.962,A -85,B 0,C 180,E1 13625.084,E2 13625.084} C_VEL
LIN {X 0,Y 344.97,Z 942.247,A -85,B 0,C 180,E1 13627.663,E2 13627.663} C_VEL
LIN {X 0,Y 346.419,Z 921.149,A -85,B 0,C 180,E1 13632.395,E2 13632.395} C_VEL
LIN {X 0,Y 367.043,Z 864.172,A -85,B 0,C 180,E1 13639.668,E2 13639.668} C_VEL
LIN {X 0,Y 382.866,Z 805.174,A -85,B 0,C 180,E1 13644.264,E2 13644.264} C_VEL
LIN {X 0,Y 370.115,Z 769.413,A -85,B 0,C 180,E1 13651.83,E2 13651.83} C_VEL
LIN {X 0,Y 361.566,Z 751.805,A -85,B 0,C 180,E1 13659.133,E2 13659.133} C_VEL
LIN {X 0,Y 360.216,Z 746.47,A -85,B 0,C 180,E1 13665.557,E2 13665.557} C_VEL
LIN {X 0,Y 365.369,Z 758.667,A -85,B 0,C 180,E1 13673.586,E2 13673.586} C_VEL
LIN {X 0,Y 374.969,Z 783.496,A -85,B 0,C 180,E1 13680.621,E2 13680.621} C_VEL
LIN {X 0,Y 380.38,Z 810.119,A -85,B 0,C 180,E1 13685.391,E2 13685.391} C_VEL
LIN {X 0,Y 361.486,Z 869.376,A -85,B 0,C 180,E1 13690.915,E2 13690.915} C_VEL
LIN {X 0,Y 341.447,Z 919.931,A -85,B 0,C 180,E1 13698.943,E2 13698.943} C_VEL
LIN {X 0,Y 325.637,Z 958.731,A -85,B 0,C 180,E1 13709.325,E2 13709.325} C_VEL
LIN {X 0,Y 317.212,Z 983.947,A -85,B 0,C 180,E1 13721.191,E2 13721.191} C_VEL
LIN {X 0,Y 314.596,Z 994.322,A -85,B 0,C 180,E1 13731.338,E2 13731.338} C_VEL
LIN {X 0,Y 314.505,Z 994.919,A -85,B 0,C 180,E1 13743.256,E2 13743.256} C_VEL
LIN {X 0,Y 317.461,Z 983.346,A -85,B 0,C 180,E1 13754.758,E2 13754.758} C_VEL
LIN {X 0,Y 325.284,Z 957.834,A -85,B 0,C 180,E1 13766.506,E2 13766.506} C_VEL
LIN {X 0,Y 340.569,Z 918.828,A -85,B 0,C 180,E1 13776.719,E2 13776.719} C_VEL
LIN {X 0,Y 359.487,Z 868.042,A -85,B 0,C 180,E1 13784.674,E2 13784.674} C_VEL
LIN {X 0,Y 377.538,Z 805.713,A -85,B 0,C 180,E1 13790.431,E2 13790.431} C_VEL
LIN {X 0,Y 360.727,Z 763.148,A -85,B 0,C 180,E1 13798.356,E2 13798.356} C_VEL
LIN {X 0,Y 338.287,Z 726.349,A -85,B 0,C 180,E1 13808.032,E2 13808.032} C_VEL
LIN {X 0,Y 318.019,Z 698.868,A -85,B 0,C 180,E1 13819.184,E2 13819.184} C_VEL
LIN {X 0,Y 313.036,Z 691.44,A -85,B 0,C 180,E1 13823.982,E2 13823.982} C_VEL
LIN {X 0,Y 313.337,Z 691.44,A -85,B 0,C 180,E1 13835.661,E2 13835.661} C_VEL
LIN {X 0,Y 314.383,Z 691.44,A -85,B 0,C 180,E1 13847.424,E2 13847.424} C_VEL
LIN {X 0,Y 315.04,Z 691.44,A -85,B 0,C 180,E1 13859.072,E2 13859.072} C_VEL
LIN {X 0,Y 314.924,Z 693.444,A -85,B 0,C 180,E1 13865.671,E2 13865.671} C_VEL
LIN {X 0,Y 331.199,Z 714.878,A -85,B 0,C 180,E1 13875.666,E2 13875.666} C_VEL
LIN {X 0,Y 355.723,Z 751.726,A -85,B 0,C 180,E1 13886.148,E2 13886.148} C_VEL
LIN {X 0,Y 377.684,Z 797.441,A -85,B 0,C 180,E1 13894.822,E2 13894.822} C_VEL
LIN {X 0,Y 380.286,Z 809.702,A -85,B 0,C 180,E1 13896.458,E2 13896.458} C_VEL
LIN {X 0,Y 362.722,Z 873.568,A -85,B 0,C 180,E1 13901.457,E2 13901.457} C_VEL
LIN {X 0,Y 343.806,Z 927.835,A -85,B 0,C 180,E1 13908.852,E2 13908.852} C_VEL
LIN {X 0,Y 327.765,Z 970.866,A -85,B 0,C 180,E1 13918.545,E2 13918.545} C_VEL
LIN {X 0,Y 318.043,Z 1001.787,A -85,B 0,C 180,E1 13930.486,E2 13930.486} C_VEL
LIN {X 0,Y 315.216,Z 1016.615,A -85,B 0,C 180,E1 13941.694,E2 13941.694} C_VEL
LIN {X 0,Y 315.346,Z 1019.666,A -85,B 0,C 180,E1 13951.378,E2 13951.378} C_VEL
LIN {X 0,Y 315.636,Z 1012.278,A -85,B 0,C 180,E1 13962.494,E2 13962.494} C_VEL
LIN {X 0,Y 321.005,Z 990.976,A -85,B 0,C 180,E1 13974.434,E2 13974.434} C_VEL
LIN {X 0,Y 333.708,Z 954.704,A -85,B 0,C 180,E1 13985.66,E2 13985.66} C_VEL
LIN {X 0,Y 346.419,Z 921.149,A -85,B 0,C 180,E1 13992.395,E2 13992.395} C_VEL
LIN {X 0,Y 349.418,Z 897.971,A -85,B 0,C 180,E1 13996.797,E2 13996.797} C_VEL
LIN {X 0,Y 370.821,Z 835.844,A -85,B 0,C 180,E1 14003.119,E2 14003.119} C_VEL
LIN {X 0,Y 377.507,Z 808.715,A -85,B 0,C 180,E1 14005.097,E2 14005.097} C_VEL
LIN {X 0,Y 366.145,Z 774.53,A -85,B 0,C 180,E1 14012.74,E2 14012.74} C_VEL
LIN {X 0,Y 358.943,Z 758.776,A -85,B 0,C 180,E1 14019.944,E2 14019.944} C_VEL
LIN {X 0,Y 358.231,Z 754.329,A -85,B 0,C 180,E1 14025.655,E2 14025.655} C_VEL
LIN {X 0,Y 362.757,Z 766.584,A -85,B 0,C 180,E1 14033.51,E2 14033.51} C_VEL
LIN {X 0,Y 371.333,Z 791.714,A -85,B 0,C 180,E1 14040.627,E2 14040.627} C_VEL
LIN {X 0,Y 374.597,Z 814.614,A -85,B 0,C 180,E1 14044.674,E2 14044.674} C_VEL
LIN {X 0,Y 354.895,Z 873.092,A -85,B 0,C 180,E1 14050.339,E2 14050.339} C_VEL
LIN {X 0,Y 333.269,Z 924.724,A -85,B 0,C 180,E1 14058.961,E2 14058.961} C_VEL
LIN {X 0,Y 316.559,Z 963.562,A -85,B 0,C 180,E1 14070.252,E2 14070.252} C_VEL
LIN {X 0,Y 309.147,Z 985.391,A -85,B 0,C 180,E1 14081.538,E2 14081.538} C_VEL
LIN {X 0,Y 306.513,Z 994.987,A -85,B 0,C 180,E1 14091.766,E2 14091.766} C_VEL
LIN {X 0,Y 306.208,Z 995.754,A -85,B 0,C 180,E1 14101.913,E2 14101.913} C_VEL
LIN {X 0,Y 308.991,Z 986.177,A -85,B 0,C 180,E1 14113.348,E2 14113.348} C_VEL
LIN {X 0,Y 316.031,Z 963.56,A -85,B 0,C 180,E1 14125.181,E2 14125.181} C_VEL
LIN {X 0,Y 331.592,Z 925.272,A -85,B 0,C 180,E1 14136.241,E2 14136.241} C_VEL
LIN {X 0,Y 350.675,Z 876.458,A -85,B 0,C 180,E1 14144.57,E2 14144.57} C_VEL
LIN {X 0,Y 369.676,Z 817.103,A -85,B 0,C 180,E1 14150.535,E2 14150.535} C_VEL
LIN {X 0,Y 370.592,Z 805.541,A -85,B 0,C 180,E1 14151.776,E2 14151.776} C_VEL
LIN {X 0,Y 353.517,Z 763.332,A -85,B 0,C 180,E1 14160.176,E2 14160.176} C_VEL
LIN {X 0,Y 331.629,Z 727.476,A -85,B 0,C 180,E1 14170.438,E2 14170.438} C_VEL
LIN {X 0,Y 314.793,Z 705.629,A -85,B 0,C 180,E1 14180.559,E2 14180.559} C_VEL
LIN {X 0,Y 308.409,Z 697.947,A -85,B 0,C 180,E1 14186.008,E2 14186.008} C_VEL
LIN {X 0,Y 305.14,Z 691.44,A -85,B 0,C 180,E1 14191.775,E2 14191.775} C_VEL
LIN {X 0,Y 306.172,Z 691.44,A -85,B 0,C 180,E1 14205.144,E2 14205.144} C_VEL
LIN {X 0,Y 306.848,Z 691.44,A -85,B 0,C 180,E1 14215.714,E2 14215.714} C_VEL
LIN {X 0,Y 307.464,Z 693.755,A -85,B 0,C 180,E1 14219.879,E2 14219.879} C_VEL
LIN {X 0,Y 318.849,Z 708.552,A -85,B 0,C 180,E1 14229.363,E2 14229.363} C_VEL
LIN {X 0,Y 339.084,Z 737.123,A -85,B 0,C 180,E1 14240.088,E2 14240.088} C_VEL
LIN {X 0,Y 361.166,Z 775.952,A -85,B 0,C 180,E1 14249.436,E2 14249.436} C_VEL
LIN {X 0,Y 374.838,Z 811.212,A -85,B 0,C 180,E1 14255.6,E2 14255.6} C_VEL
LIN {X 0,Y 356.514,Z 875.018,A -85,B 0,C 180,E1 14260.689,E2 14260.689} C_VEL
LIN {X 0,Y 336.944,Z 928.695,A -85,B 0,C 180,E1 14268.169,E2 14268.169} C_VEL
LIN {X 0,Y 320.04,Z 971.939,A -85,B 0,C 180,E1 14278.23,E2 14278.23} C_VEL
LIN {X 0,Y 310.288,Z 1001.438,A -85,B 0,C 180,E1 14289.978,E2 14289.978} C_VEL
LIN {X 0,Y 307.229,Z 1016.437,A -85,B 0,C 180,E1 14301.646,E2 14301.646} C_VEL
LIN {X 0,Y 307.34,Z 1019.365,A -85,B 0,C 180,E1 14311.413,E2 14311.413} C_VEL
LIN {X 0,Y 307.706,Z 1011.972,A -85,B 0,C 180,E1 14322.822,E2 14322.822} C_VEL
LIN {X 0,Y 313.412,Z 990.781,A -85,B 0,C 180,E1 14335.017,E2 14335.017} C_VEL
LIN {X 0,Y 327.151,Z 953.821,A -85,B 0,C 180,E1 14346.671,E2 14346.671} C_VEL
LIN {X 0,Y 346.328,Z 905.788,A -85,B 0,C 180,E1 14355.699,E2 14355.699} C_VEL
LIN {X 0,Y 349.418,Z 897.971,A -85,B 0,C 180,E1 14356.797,E2 14356.797} C_VEL
LIN {X 0,Y 353.672,Z 872.725,A -85,B 0,C 180,E1 14360.809,E2 14360.809} C_VEL
LIN {X 0,Y 372.21,Z 812.488,A -85,B 0,C 180,E1 14365.9,E2 14365.9} C_VEL
LIN {X 0,Y 362.392,Z 780.404,A -85,B 0,C 180,E1 14373.471,E2 14373.471} C_VEL
LIN {X 0,Y 356.27,Z 765.61,A -85,B 0,C 180,E1 14380.759,E2 14380.759} C_VEL
LIN {X 0,Y 355.998,Z 762.337,A -85,B 0,C 180,E1 14385.677,E2 14385.677} C_VEL
LIN {X 0,Y 359.832,Z 774.041,A -85,B 0,C 180,E1 14393.283,E2 14393.283} C_VEL
LIN {X 0,Y 367.489,Z 799.807,A -85,B 0,C 180,E1 14400.619,E2 14400.619} C_VEL
LIN {X 0,Y 369.232,Z 818.079,A -85,B 0,C 180,E1 14403.856,E2 14403.856} C_VEL
LIN {X 0,Y 349.229,Z 874.456,A -85,B 0,C 180,E1 14409.449,E2 14409.449} C_VEL
LIN {X 0,Y 326.74,Z 925.615,A -85,B 0,C 180,E1 14418.147,E2 14418.147} C_VEL
LIN {X 0,Y 309.682,Z 963.083,A -85,B 0,C 180,E1 14429.213,E2 14429.213} C_VEL
LIN {X 0,Y 301.195,Z 986.189,A -85,B 0,C 180,E1 14441.461,E2 14441.461} C_VEL
LIN {X 0,Y 298.449,Z 995.559,A -85,B 0,C 180,E1 14452.051,E2 14452.051} C_VEL
LIN {X 0,Y 298.6,Z 995.019,A -85,B 0,C 180,E1 14464.407,E2 14464.407} C_VEL
LIN {X 0,Y 301.913,Z 983.025,A -85,B 0,C 180,E1 14476.188,E2 14476.188} C_VEL
LIN {X 0,Y 311.324,Z 956.944,A -85,B 0,C 180,E1 14488.417,E2 14488.417} C_VEL
LIN {X 0,Y 328.648,Z 916.79,A -85,B 0,C 180,E1 14498.967,E2 14498.967} C_VEL
LIN {X 0,Y 349.301,Z 865.045,A -85,B 0,C 180,E1 14506.948,E2 14506.948} C_VEL
LIN {X 0,Y 365.308,Z 811.305,A -85,B 0,C 180,E1 14512.107,E2 14512.107} C_VEL
LIN {X 0,Y 350.302,Z 771.641,A -85,B 0,C 180,E1 14520.179,E2 14520.179} C_VEL
LIN {X 0,Y 330.437,Z 737.019,A -85,B 0,C 180,E1 14530.071,E2 14530.071} C_VEL
LIN {X 0,Y 313.418,Z 713.494,A -85,B 0,C 180,E1 14540.663,E2 14540.663} C_VEL
LIN {X 0,Y 302.873,Z 699.118,A -85,B 0,C 180,E1 14551.545,E2 14551.545} C_VEL
LIN {X 0,Y 299.536,Z 695.611,A -85,B 0,C 180,E1 14568.646,E2 14568.646} C_VEL
LIN {X 0,Y 306.126,Z 701.78,A -85,B 0,C 180,E1 14579.701,E2 14579.701} C_VEL
LIN {X 0,Y 317.31,Z 716.685,A -85,B 0,C 180,E1 14589.167,E2 14589.167} C_VEL
LIN {X 0,Y 336.268,Z 744.216,A -85,B 0,C 180,E1 14599.666,E2 14599.666} C_VEL
LIN {X 0,Y 356.963,Z 782.102,A -85,B 0,C 180,E1 14608.968,E2 14608.968} C_VEL
LIN {X 0,Y 368.735,Z 815.204,A -85,B 0,C 180,E1 14614.878,E2 14614.878} C_VEL
LIN {X 0,Y 349.688,Z 878.337,A -85,B 0,C 180,E1 14620.1,E2 14620.1} C_VEL
LIN {X 0,Y 328.946,Z 932.559,A -85,B 0,C 180,E1 14628.012,E2 14628.012} C_VEL
LIN {X 0,Y 311.836,Z 974.274,A -85,B 0,C 180,E1 14638.308,E2 14638.308} C_VEL
LIN {X 0,Y 302.155,Z 1002.427,A -85,B 0,C 180,E1 14650.181,E2 14650.181} C_VEL
LIN {X 0,Y 299.188,Z 1016.918,A -85,B 0,C 180,E1 14662.713,E2 14662.713} C_VEL
LIN {X 0,Y 299.333,Z 1019.065,A -85,B 0,C 180,E1 14671.451,E2 14671.451} C_VEL
LIN {X 0,Y 299.784,Z 1011.67,A -85,B 0,C 180,E1 14683.166,E2 14683.166} C_VEL
LIN {X 0,Y 305.867,Z 990.594,A -85,B 0,C 180,E1 14695.628,E2 14695.628} C_VEL
LIN {X 0,Y 320.423,Z 953.582,A -85,B 0,C 180,E1 14707.573,E2 14707.573} C_VEL
LIN {X 0,Y 340.815,Z 905.196,A -85,B 0,C 180,E1 14716.771,E2 14716.771} C_VEL
LIN {X 0,Y 353.672,Z 872.725,A -85,B 0,C 180,E1 14720.809,E2 14720.809} C_VEL
LIN {X 0,Y 358.412,Z 845.693,A -85,B 0,C 180,E1 14724.435,E2 14724.435} C_VEL
LIN {X 0,Y 366.788,Z 815.39,A -85,B 0,C 180,E1 14726.912,E2 14726.912} C_VEL
LIN {X 0,Y 358.479,Z 785.611,A -85,B 0,C 180,E1 14734.391,E2 14734.391} C_VEL
LIN {X 0,Y 353.585,Z 772.073,A -85,B 0,C 180,E1 14741.905,E2 14741.905} C_VEL
LIN {X 0,Y 353.585,Z 770.653,A -85,B 0,C 180,E1 14746.035,E2 14746.035} C_VEL
LIN {X 0,Y 356.934,Z 781.782,A -85,B 0,C 180,E1 14753.228,E2 14753.228} C_VEL
LIN {X 0,Y 363.414,Z 807.959,A -85,B 0,C 180,E1 14760.626,E2 14760.626} C_VEL
LIN {X 0,Y 363.996,Z 821.57,A -85,B 0,C 180,E1 14763.014,E2 14763.014} C_VEL
LIN {X 0,Y 342.273,Z 879.092,A -85,B 0,C 180,E1 14768.955,E2 14768.955} C_VEL
LIN {X 0,Y 319.966,Z 927.188,A -85,B 0,C 180,E1 14777.456,E2 14777.456} C_VEL
LIN {X 0,Y 302.375,Z 963.757,A -85,B 0,C 180,E1 14788.564,E2 14788.564} C_VEL
LIN {X 0,Y 293.258,Z 986.994,A -85,B 0,C 180,E1 14801.38,E2 14801.38} C_VEL
LIN {X 0,Y 290.24,Z 996.263,A -85,B 0,C 180,E1 14813.038,E2 14813.038} C_VEL
LIN {X 0,Y 290.959,Z 994.511,A -85,B 0,C 180,E1 14825.944,E2 14825.944} C_VEL
LIN {X 0,Y 294.501,Z 981.814,A -85,B 0,C 180,E1 14837.655,E2 14837.655} C_VEL
LIN {X 0,Y 304.779,Z 955.653,A -85,B 0,C 180,E1 14849.691,E2 14849.691} C_VEL
LIN {X 0,Y 323.491,Z 914.492,A -85,B 0,C 180,E1 14860.4,E2 14860.4} C_VEL
LIN {X 0,Y 345.087,Z 861.643,A -85,B 0,C 180,E1 14868.356,E2 14868.356} C_VEL
LIN {X 0,Y 359.387,Z 814.483,A -85,B 0,C 180,E1 14872.911,E2 14872.911} C_VEL
LIN {X 0,Y 345.39,Z 776.23,A -85,B 0,C 180,E1 14881.008,E2 14881.008} C_VEL
LIN {X 0,Y 326.048,Z 741.578,A -85,B 0,C 180,E1 14891.381,E2 14891.381} C_VEL
LIN {X 0,Y 310.578,Z 720.186,A -85,B 0,C 180,E1 14901.775,E2 14901.775} C_VEL
LIN {X 0,Y 301.193,Z 706.853,A -85,B 0,C 180,E1 14912.318,E2 14912.318} C_VEL
LIN {X 0,Y 298.392,Z 703.521,A -85,B 0,C 180,E1 14928.602,E2 14928.602} C_VEL
LIN {X 0,Y 304.803,Z 709.712,A -85,B 0,C 180,E1 14939.521,E2 14939.521} C_VEL
LIN {X 0,Y 316.078,Z 725.384,A -85,B 0,C 180,E1 14949.276,E2 14949.276} C_VEL
LIN {X 0,Y 334.028,Z 752.269,A -85,B 0,C 180,E1 14959.557,E2 14959.557} C_VEL
LIN {X 0,Y 353.912,Z 790.999,A -85,B 0,C 180,E1 14969.118,E2 14969.118} C_VEL
LIN {X 0,Y 362.679,Z 819.553,A -85,B 0,C 180,E1 14974.17,E2 14974.17} C_VEL
LIN {X 0,Y 342.939,Z 881.217,A -85,B 0,C 180,E1 14979.461,E2 14979.461} C_VEL
LIN {X 0,Y 321.986,Z 933.713,A -85,B 0,C 180,E1 14987.348,E2 14987.348} C_VEL
LIN {X 0,Y 303.69,Z 976.467,A -85,B 0,C 180,E1 14998.35,E2 14998.35} C_VEL
LIN {X 0,Y 293.559,Z 1004.447,A -85,B 0,C 180,E1 15011.148,E2 15011.148} C_VEL
LIN {X 0,Y 291.201,Z 1016.605,A -85,B 0,C 180,E1 15022.512,E2 15022.512} C_VEL
LIN {X 0,Y 291.331,Z 1018.765,A -85,B 0,C 180,E1 15031.491,E2 15031.491} C_VEL
LIN {X 0,Y 291.872,Z 1011.373,A -85,B 0,C 180,E1 15043.53,E2 15043.53} C_VEL
LIN {X 0,Y 298.613,Z 989.642,A -85,B 0,C 180,E1 15056.607,E2 15056.607} C_VEL
LIN {X 0,Y 314.253,Z 952.4,A -85,B 0,C 180,E1 15068.756,E2 15068.756} C_VEL
LIN {X 0,Y 336.234,Z 902.856,A -85,B 0,C 180,E1 15078.134,E2 15078.134} C_VEL
LIN {X 0,Y 358.412,Z 845.693,A -85,B 0,C 180,E1 15084.435,E2 15084.435} C_VEL
LIN {X 0,Y 360.074,Z 827.551,A -85,B 0,C 180,E1 15086.927,E2 15086.927} C_VEL
LIN {X 0,Y 361.478,Z 817.867,A -85,B 0,C 180,E1 15088.045,E2 15088.045} C_VEL
LIN {X 0,Y 354.659,Z 790.774,A -85,B 0,C 180,E1 15095.379,E2 15095.379} C_VEL
LIN {X 0,Y 351.233,Z 777.23,A -85,B 0,C 180,E1 15103.723,E2 15103.723} C_VEL
LIN {X 0,Y 353.15,Z 786.64,A -85,B 0,C 180,E1 15112.002,E2 15112.002} C_VEL
LIN {X 0,Y 358.179,Z 809.28,A -85,B 0,C 180,E1 15119.118,E2 15119.118} C_VEL
LIN {X 0,Y 358.841,Z 824.89,A -85,B 0,C 180,E1 15122.136,E2 15122.136} C_VEL
LIN {X 0,Y 335.606,Z 883.186,A -85,B 0,C 180,E1 15128.367,E2 15128.367} C_VEL
LIN {X 0,Y 311.655,Z 931.804,A -85,B 0,C 180,E1 15137.465,E2 15137.465} C_VEL
LIN {X 0,Y 294.147,Z 966.369,A -85,B 0,C 180,E1 15148.702,E2 15148.702} C_VEL
LIN {X 0,Y 285.181,Z 988.321,A -85,B 0,C 180,E1 15161.731,E2 15161.731} C_VEL
LIN {X 0,Y 282.385,Z 996.247,A -85,B 0,C 180,E1 15171.829,E2 15171.829} C_VEL
LIN {X 0,Y 282.225,Z 996.435,A -85,B 0,C 180,E1 15182.804,E2 15182.804} C_VEL
LIN {X 0,Y 285.487,Z 986.896,A -85,B 0,C 180,E1 15194.666,E2 15194.666} C_VEL
LIN {X 0,Y 294.526,Z 963.053,A -85,B 0,C 180,E1 15207.787,E2 15207.787} C_VEL
LIN {X 0,Y 313.016,Z 923.89,A -85,B 0,C 180,E1 15219.419,E2 15219.419} C_VEL
LIN {X 0,Y 335.347,Z 872.894,A -85,B 0,C 180,E1 15228.039,E2 15228.039} C_VEL
LIN {X 0,Y 353.56,Z 817.962,A -85,B 0,C 180,E1 15233.688,E2 15233.688} C_VEL
LIN {X 0,Y 339.775,Z 779.339,A -85,B 0,C 180,E1 15242.259,E2 15242.259} C_VEL
LIN {X 0,Y 322.003,Z 747.174,A -85,B 0,C 180,E1 15252.45,E2 15252.45} C_VEL
LIN {X 0,Y 307.91,Z 726.619,A -85,B 0,C 180,E1 15262.871,E2 15262.871} C_VEL
LIN {X 0,Y 299.146,Z 714.347,A -85,B 0,C 180,E1 15273.687,E2 15273.687} C_VEL
LIN {X 0,Y 297.353,Z 711.564,A -85,B 0,C 180,E1 15288.935,E2 15288.935} C_VEL
LIN {X 0,Y 303.545,Z 717.747,A -85,B 0,C 180,E1 15299.43,E2 15299.43} C_VEL
LIN {X 0,Y 317.244,Z 736.723,A -85,B 0,C 180,E1 15310.995,E2 15310.995} C_VEL
LIN {X 0,Y 337.418,Z 770.918,A -85,B 0,C 180,E1 15322.519,E2 15322.519} C_VEL
LIN {X 0,Y 355.357,Z 812.935,A -85,B 0,C 180,E1 15331.861,E2 15331.861} C_VEL
LIN {X 0,Y 356.453,Z 824.393,A -85,B 0,C 180,E1 15333.466,E2 15333.466} C_VEL
LIN {X 0,Y 335.429,Z 886.357,A -85,B 0,C 180,E1 15339.075,E2 15339.075} C_VEL
LIN {X 0,Y 313.554,Z 938.084,A -85,B 0,C 180,E1 15347.342,E2 15347.342} C_VEL
LIN {X 0,Y 295.662,Z 978.216,A -85,B 0,C 180,E1 15358.282,E2 15358.282} C_VEL
LIN {X 0,Y 285.414,Z 1005.277,A -85,B 0,C 180,E1 15371.394,E2 15371.394} C_VEL
LIN {X 0,Y 283.213,Z 1016.289,A -85,B 0,C 180,E1 15382.3,E2 15382.3} C_VEL
LIN {X 0,Y 283.324,Z 1018.466,A -85,B 0,C 180,E1 15391.533,E2 15391.533} C_VEL
LIN {X 0,Y 284.001,Z 1011.081,A -85,B 0,C 180,E1 15403.912,E2 15403.912} C_VEL
LIN {X 0,Y 291.128,Z 989.371,A -85,B 0,C 180,E1 15417.347,E2 15417.347} C_VEL
LIN {X 0,Y 308.131,Z 951.29,A -85,B 0,C 180,E1 15429.984,E2 15429.984} C_VEL
LIN {X 0,Y 331.463,Z 901.423,A -85,B 0,C 180,E1 15439.412,E2 15439.412} C_VEL
LIN {X 0,Y 355.282,Z 841.87,A -85,B 0,C 180,E1 15445.852,E2 15445.852} C_VEL
LIN {X 0,Y 360.074,Z 827.551,A -85,B 0,C 180,E1 15446.927,E2 15446.927} C_VEL
LIN {X 0,Y 358.97,Z 820.831,A -85,B 0,C 180,E1 15448.347,E2 15448.347} C_VEL
LIN {X 0,Y 355.499,Z 816.113,A -85,B 0,C 180,E1 15450.226,E2 15450.226} C_VEL
LIN {X 0,Y 350.111,Z 793.875,A -85,B 0,C 180,E1 15457.395,E2 15457.395} C_VEL
LIN {X 0,Y 348.475,Z 785.167,A -85,B 0,C 180,E1 15463.591,E2 15463.591} C_VEL
LIN {X 0,Y 350.008,Z 794.583,A -85,B 0,C 180,E1 15472.083,E2 15472.083} C_VEL
LIN {X 0,Y 354.019,Z 818.479,A -85,B 0,C 180,E1 15479.415,E2 15479.415} C_VEL
LIN {X 0,Y 353.328,Z 829.474,A -85,B 0,C 180,E1 15481.342,E2 15481.342} C_VEL
LIN {X 0,Y 329.218,Z 886.595,A -85,B 0,C 180,E1 15487.666,E2 15487.666} C_VEL
LIN {X 0,Y 304.336,Z 934.565,A -85,B 0,C 180,E1 15497.007,E2 15497.007} C_VEL
LIN {X 0,Y 285.128,Z 970.506,A -85,B 0,C 180,E1 15509.606,E2 15509.606} C_VEL
LIN {X 0,Y 276.798,Z 990.775,A -85,B 0,C 180,E1 15523.299,E2 15523.299} C_VEL
LIN {X 0,Y 273.942,Z 997.414,A -85,B 0,C 180,E1 15534.433,E2 15534.433} C_VEL
LIN {X 0,Y 275.199,Z 994.494,A -85,B 0,C 180,E1 15547.384,E2 15547.384} C_VEL
LIN {X 0,Y 279.719,Z 980.646,A -85,B 0,C 180,E1 15559.846,E2 15559.846} C_VEL
LIN {X 0,Y 292.956,Z 951.37,A -85,B 0,C 180,E1 15572.971,E2 15572.971} C_VEL
LIN {X 0,Y 313.39,Z 910.006,A -85,B 0,C 180,E1 15583.299,E2 15583.299} C_VEL
LIN {X 0,Y 336.341,Z 856.915,A -85,B 0,C 180,E1 15590.988,E2 15590.988} C_VEL
LIN {X 0,Y 347.55,Z 820.491,A -85,B 0,C 180,E1 15594.67,E2 15594.67} C_VEL
LIN {X 0,Y 334.361,Z 782.842,A -85,B 0,C 180,E1 15603.428,E2 15603.428} C_VEL
LIN {X 0,Y 316.679,Z 749.981,A -85,B 0,C 180,E1 15614.551,E2 15614.551} C_VEL
LIN {X 0,Y 303.075,Z 729.52,A -85,B 0,C 180,E1 15626.219,E2 15626.219} C_VEL
LIN {X 0,Y 297.179,Z 721.791,A -85,B 0,C 180,E1 15634.992,E2 15634.992} C_VEL
LIN {X 0,Y 296.241,Z 719.557,A -85,B 0,C 180,E1 15649.266,E2 15649.266} C_VEL
LIN {X 0,Y 302.114,Z 725.76,A -85,B 0,C 180,E1 15659.334,E2 15659.334} C_VEL
LIN {X 0,Y 315.259,Z 745.052,A -85,B 0,C 180,E1 15670.906,E2 15670.906} C_VEL
LIN {X 0,Y 333.798,Z 777.547,A -85,B 0,C 180,E1 15682.079,E2 15682.079} C_VEL
LIN {X 0,Y 350.55,Z 819.351,A -85,B 0,C 180,E1 15691.579,E2 15691.579} C_VEL
LIN {X 0,Y 350.054,Z 829.498,A -85,B 0,C 180,E1 15692.798,E2 15692.798} C_VEL
LIN {X 0,Y 328.837,Z 888.99,A -85,B 0,C 180,E1 15698.374,E2 15698.374} C_VEL
LIN {X 0,Y 305.697,Z 941.092,A -85,B 0,C 180,E1 15707.046,E2 15707.046} C_VEL
LIN {X 0,Y 287.496,Z 980.025,A -85,B 0,C 180,E1 15718.275,E2 15718.275} C_VEL
LIN {X 0,Y 277.246,Z 1006.054,A -85,B 0,C 180,E1 15731.653,E2 15731.653} C_VEL
LIN {X 0,Y 275.241,Z 1015.972,A -85,B 0,C 180,E1 15742.076,E2 15742.076} C_VEL
LIN {X 0,Y 275.334,Z 1018.167,A -85,B 0,C 180,E1 15751.578,E2 15751.578} C_VEL
LIN {X 0,Y 276.107,Z 1010.794,A -85,B 0,C 180,E1 15764.319,E2 15764.319} C_VEL
LIN {X 0,Y 283.957,Z 988.351,A -85,B 0,C 180,E1 15778.468,E2 15778.468} C_VEL
LIN {X 0,Y 301.41,Z 951.789,A -85,B 0,C 180,E1 15790.84,E2 15790.84} C_VEL
LIN {X 0,Y 326.088,Z 901.75,A -85,B 0,C 180,E1 15800.475,E2 15800.475} C_VEL
LIN {X 0,Y 350.844,Z 842.578,A -85,B 0,C 180,E1 15806.935,E2 15806.935} C_VEL
LIN {X 0,Y 356.65,Z 822.65,A -85,B 0,C 180,E1 15808.738,E2 15808.738} C_VEL
LIN {X 0,Y 355.499,Z 816.113,A -85,B 0,C 180,E1 15810.226,E2 15810.226} C_VEL
LIN {X 0,Y 347.922,Z 805.681,A -85,B 0,C 180,E1 15815.659,E2 15815.659} C_VEL
LIN {X 0,Y 345.494,Z 793.026,A -85,B 0,C 180,E1 15823.445,E2 15823.445} C_VEL
LIN {X 0,Y 346.402,Z 800.382,A -85,B 0,C 180,E1 15831.211,E2 15831.211} C_VEL
LIN {X 0,Y 349.293,Z 822.424,A -85,B 0,C 180,E1 15838.473,E2 15838.473} C_VEL
LIN {X 0,Y 348.746,Z 831.92,A -85,B 0,C 180,E1 15840.34,E2 15840.34} C_VEL
LIN {X 0,Y 323.498,Z 888.769,A -85,B 0,C 180,E1 15846.765,E2 15846.765} C_VEL
LIN {X 0,Y 297.423,Z 936.493,A -85,B 0,C 180,E1 15856.329,E2 15856.329} C_VEL
LIN {X 0,Y 277.379,Z 972.005,A -85,B 0,C 180,E1 15869.305,E2 15869.305} C_VEL
LIN {X 0,Y 268.784,Z 991.606,A -85,B 0,C 180,E1 15883.378,E2 15883.378} C_VEL
LIN {X 0,Y 265.745,Z 997.914,A -85,B 0,C 180,E1 15895.946,E2 15895.946} C_VEL
LIN {X 0,Y 267.668,Z 993.487,A -85,B 0,C 180,E1 15909.378,E2 15909.378} C_VEL
LIN {X 0,Y 274.424,Z 976.057,A -85,B 0,C 180,E1 15923.332,E2 15923.332} C_VEL
LIN {X 0,Y 290.632,Z 943.553,A -85,B 0,C 180,E1 15936.365,E2 15936.365} C_VEL
LIN {X 0,Y 312.503,Z 899.8,A -85,B 0,C 180,E1 15946.216,E2 15946.216} C_VEL
LIN {X 0,Y 335.791,Z 845.081,A -85,B 0,C 180,E1 15953.295,E2 15953.295} C_VEL
LIN {X 0,Y 341.794,Z 824.295,A -85,B 0,C 180,E1 15955.409,E2 15955.409} C_VEL
LIN {X 0,Y 329.545,Z 787.899,A -85,B 0,C 180,E1 15964.232,E2 15964.232} C_VEL
LIN {X 0,Y 313.443,Z 756.736,A -85,B 0,C 180,E1 15975.178,E2 15975.178} C_VEL
LIN {X 0,Y 301.035,Z 737.1,A -85,B 0,C 180,E1 15986.591,E2 15986.591} C_VEL
LIN {X 0,Y 295.523,Z 729.422,A -85,B 0,C 180,E1 15995.588,E2 15995.588} C_VEL
LIN {X 0,Y 295.042,Z 727.586,A -85,B 0,C 180,E1 16009.597,E2 16009.597} C_VEL
LIN {X 0,Y 300.688,Z 733.785,A -85,B 0,C 180,E1 16019.337,E2 16019.337} C_VEL
LIN {X 0,Y 313.387,Z 753.683,A -85,B 0,C 180,E1 16031.045,E2 16031.045} C_VEL
LIN {X 0,Y 330.364,Z 784.965,A -85,B 0,C 180,E1 16041.877,E2 16041.877} C_VEL
LIN {X 0,Y 345.817,Z 826.421,A -85,B 0,C 180,E1 16051.44,E2 16051.44} C_VEL
LIN {X 0,Y 323.613,Z 888.278,A -85,B 0,C 180,E1 16057.237,E2 16057.237} C_VEL
LIN {X 0,Y 299.47,Z 940.698,A -85,B 0,C 180,E1 16066.006,E2 16066.006} C_VEL
LIN {X 0,Y 279.949,Z 980.542,A -85,B 0,C 180,E1 16077.762,E2 16077.762} C_VEL
LIN {X 0,Y 269.48,Z 1005.696,A -85,B 0,C 180,E1 16091.105,E2 16091.105} C_VEL
LIN {X 0,Y 267.097,Z 1016.502,A -85,B 0,C 180,E1 16103.419,E2 16103.419} C_VEL
LIN {X 0,Y 267.16,Z 1017.127,A -85,B 0,C 180,E1 16114.886,E2 16114.886} C_VEL
LIN {X 0,Y 269.275,Z 1006.809,A -85,B 0,C 180,E1 16128.056,E2 16128.056} C_VEL
LIN {X 0,Y 278.927,Z 982.799,A -85,B 0,C 180,E1 16141.686,E2 16141.686} C_VEL
LIN {X 0,Y 299.673,Z 943.204,A -85,B 0,C 180,E1 16153.976,E2 16153.976} C_VEL
LIN {X 0,Y 325.482,Z 892.735,A -85,B 0,C 180,E1 16162.857,E2 16162.857} C_VEL
LIN {X 0,Y 350.883,Z 831.747,A -85,B 0,C 180,E1 16168.94,E2 16168.94} C_VEL
LIN {X 0,Y 350.245,Z 817.275,A -85,B 0,C 180,E1 16171.965,E2 16171.965} C_VEL
LIN {X 0,Y 347.922,Z 805.681,A -85,B 0,C 180,E1 16175.659,E2 16175.659} C_VEL
LIN {X 0,Y 342.394,Z 802.767,A -85,B 0,C 180,E1 16181.51,E2 16181.51} C_VEL
LIN {X 0,Y 342.188,Z 802.237,A -85,B 0,C 180,E1 16187.222,E2 16187.222} C_VEL
LIN {X 0,Y 343.889,Z 815.744,A -85,B 0,C 180,E1 16194.384,E2 16194.384} C_VEL
LIN {X 0,Y 343.865,Z 835.515,A -85,B 0,C 180,E1 16199.397,E2 16199.397} C_VEL
LIN {X 0,Y 317.205,Z 892.19,A -85,B 0,C 180,E1 16206.011,E2 16206.011} C_VEL
LIN {X 0,Y 290.611,Z 938.297,A -85,B 0,C 180,E1 16215.589,E2 16215.589} C_VEL
LIN {X 0,Y 270.075,Z 972.642,A -85,B 0,C 180,E1 16228.565,E2 16228.565} C_VEL
LIN {X 0,Y 261.221,Z 991.123,A -85,B 0,C 180,E1 16241.96,E2 16241.96} C_VEL
LIN {X 0,Y 258.175,Z 997.581,A -85,B 0,C 180,E1 16252.564,E2 16252.564} C_VEL
LIN {X 0,Y 258.671,Z 996.355,A -85,B 0,C 180,E1 16265.48,E2 16265.48} C_VEL
LIN {X 0,Y 262.906,Z 984.972,A -85,B 0,C 180,E1 16278.346,E2 16278.346} C_VEL
LIN {X 0,Y 275.658,Z 958.57,A -85,B 0,C 180,E1 16292.368,E2 16292.368} C_VEL
LIN {X 0,Y 297.349,Z 918.664,A -85,B 0,C 180,E1 16303.723,E2 16303.723} C_VEL
LIN {X 0,Y 321.817,Z 867.525,A -85,B 0,C 180,E1 16311.983,E2 16311.983} C_VEL
LIN {X 0,Y 336.011,Z 828.003,A -85,B 0,C 180,E1 16316.188,E2 16316.188} C_VEL
LIN {X 0,Y 324.737,Z 792.736,A -85,B 0,C 180,E1 16325.098,E2 16325.098} C_VEL
LIN {X 0,Y 309.784,Z 762.937,A -85,B 0,C 180,E1 16336.047,E2 16336.047} C_VEL
LIN {X 0,Y 298.659,Z 744.424,A -85,B 0,C 180,E1 16347.217,E2 16347.217} C_VEL
LIN {X 0,Y 293.882,Z 737.264,A -85,B 0,C 180,E1 16355.566,E2 16355.566} C_VEL
LIN {X 0,Y 293.487,Z 735.429,A -85,B 0,C 180,E1 16369.541,E2 16369.541} C_VEL
LIN {X 0,Y 298.992,Z 741.749,A -85,B 0,C 180,E1 16379.333,E2 16379.333} C_VEL
LIN {X 0,Y 311.198,Z 761.8,A -85,B 0,C 180,E1 16391.035,E2 16391.035} C_VEL
LIN {X 0,Y 326.96,Z 792.712,A -85,B 0,C 180,E1 16401.758,E2 16401.758} C_VEL
LIN {X 0,Y 340.067,Z 830.664,A -85,B 0,C 180,E1 16410.725,E2 16410.725} C_VEL
LIN {X 0,Y 317.009,Z 890.924,A -85,B 0,C 180,E1 16416.503,E2 16416.503} C_VEL
LIN {X 0,Y 292.099,Z 942.715,A -85,B 0,C 180,E1 16425.46,E2 16425.46} C_VEL
LIN {X 0,Y 271.497,Z 982.807,A -85,B 0,C 180,E1 16437.924,E2 16437.924} C_VEL
LIN {X 0,Y 261.316,Z 1006.325,A -85,B 0,C 180,E1 16451.371,E2 16451.371} C_VEL
LIN {X 0,Y 259.142,Z 1016.811,A -85,B 0,C 180,E1 16464.959,E2 16464.959} C_VEL
LIN {X 0,Y 259.172,Z 1016.834,A -85,B 0,C 180,E1 16475.037,E2 16475.037} C_VEL
LIN {X 0,Y 261.459,Z 1006.54,A -85,B 0,C 180,E1 16488.615,E2 16488.615} C_VEL
LIN {X 0,Y 272.478,Z 981.391,A -85,B 0,C 180,E1 16503.113,E2 16503.113} C_VEL
LIN {X 0,Y 295.507,Z 940.134,A -85,B 0,C 180,E1 16515.828,E2 16515.828} C_VEL
LIN {X 0,Y 323.469,Z 887.364,A -85,B 0,C 180,E1 16524.765,E2 16524.765} C_VEL
LIN {X 0,Y 346.827,Z 830.56,A -85,B 0,C 180,E1 16530.552,E2 16530.552} C_VEL
LIN {X 0,Y 343.342,Z 807.983,A -85,B 0,C 180,E1 16537.969,E2 16537.969} C_VEL
LIN {X 0,Y 342.394,Z 802.767,A -85,B 0,C 180,E1 16541.51,E2 16541.51} C_VEL
LIN {X 0,Y 338.868,Z 809.795,A -85,B 0,C 180,E1 16547.402,E2 16547.402} C_VEL
LIN {X 0,Y 339.817,Z 823.275,A -85,B 0,C 180,E1 16554.316,E2 16554.316} C_VEL
LIN {X 0,Y 338.72,Z 839.948,A -85,B 0,C 180,E1 16558.506,E2 16558.506} C_VEL
LIN {X 0,Y 310.842,Z 895.995,A -85,B 0,C 180,E1 16565.283,E2 16565.283} C_VEL
LIN {X 0,Y 282.64,Z 942.048,A -85,B 0,C 180,E1 16575.372,E2 16575.372} C_VEL
LIN {X 0,Y 262.373,Z 974.028,A -85,B 0,C 180,E1 16588.21,E2 16588.21} C_VEL
LIN {X 0,Y 253.361,Z 991.559,A -85,B 0,C 180,E1 16601.522,E2 16601.522} C_VEL
LIN {X 0,Y 249.796,Z 998.479,A -85,B 0,C 180,E1 16615.152,E2 16615.152} C_VEL
LIN {X 0,Y 251.619,Z 994.566,A -85,B 0,C 180,E1 16629.28,E2 16629.28} C_VEL
LIN {X 0,Y 258.778,Z 977.922,A -85,B 0,C 180,E1 16643.964,E2 16643.964} C_VEL
LIN {X 0,Y 275.658,Z 947.128,A -85,B 0,C 180,E1 16657.368,E2 16657.368} C_VEL
LIN {X 0,Y 299.207,Z 904.233,A -85,B 0,C 180,E1 16667.719,E2 16667.719} C_VEL
LIN {X 0,Y 324.846,Z 848.462,A -85,B 0,C 180,E1 16675.234,E2 16675.234} C_VEL
LIN {X 0,Y 330.35,Z 831.951,A -85,B 0,C 180,E1 16676.938,E2 16676.938} C_VEL
LIN {X 0,Y 319.928,Z 797.609,A -85,B 0,C 180,E1 16685.956,E2 16685.956} C_VEL
LIN {X 0,Y 306.057,Z 768.881,A -85,B 0,C 180,E1 16697.034,E2 16697.034} C_VEL
LIN {X 0,Y 296.054,Z 751.725,A -85,B 0,C 180,E1 16707.923,E2 16707.923} C_VEL
LIN {X 0,Y 291.827,Z 744.799,A -85,B 0,C 180,E1 16716.374,E2 16716.374} C_VEL
LIN {X 0,Y 292,Z 743.442,A -85,B 0,C 180,E1 16730.01,E2 16730.01} C_VEL
LIN {X 0,Y 297.052,Z 749.558,A -85,B 0,C 180,E1 16739.191,E2 16739.191} C_VEL
LIN {X 0,Y 308.388,Z 769.227,A -85,B 0,C 180,E1 16750.778,E2 16750.778} C_VEL
LIN {X 0,Y 322.955,Z 799.411,A -85,B 0,C 180,E1 16761.41,E2 16761.41} C_VEL
LIN {X 0,Y 334.397,Z 833.53,A -85,B 0,C 180,E1 16769.785,E2 16769.785} C_VEL
LIN {X 0,Y 310.127,Z 894.15,A -85,B 0,C 180,E1 16775.819,E2 16775.819} C_VEL
LIN {X 0,Y 285.33,Z 943.49,A -85,B 0,C 180,E1 16784.626,E2 16784.626} C_VEL
LIN {X 0,Y 264.5,Z 982.309,A -85,B 0,C 180,E1 16796.969,E2 16796.969} C_VEL
LIN {X 0,Y 252.981,Z 1007.421,A -85,B 0,C 180,E1 16812.064,E2 16812.064} C_VEL
LIN {X 0,Y 251.143,Z 1016.538,A -85,B 0,C 180,E1 16824.943,E2 16824.943} C_VEL
LIN {X 0,Y 251.162,Z 1016.544,A -85,B 0,C 180,E1 16835.199,E2 16835.199} C_VEL
LIN {X 0,Y 253.616,Z 1006.277,A -85,B 0,C 180,E1 16849.213,E2 16849.213} C_VEL
LIN {X 0,Y 264.899,Z 982.367,A -85,B 0,C 180,E1 16863.597,E2 16863.597} C_VEL
LIN {X 0,Y 288.548,Z 942.193,A -85,B 0,C 180,E1 16876.516,E2 16876.516} C_VEL
LIN {X 0,Y 316.877,Z 891.706,A -85,B 0,C 180,E1 16885.456,E2 16885.456} C_VEL
LIN {X 0,Y 342.082,Z 835.173,A -85,B 0,C 180,E1 16891.347,E2 16891.347} C_VEL
LIN {X 0,Y 339.683,Z 814.394,A -85,B 0,C 180,E1 16898.555,E2 16898.555} C_VEL
LIN {X 0,Y 338.978,Z 808.12,A -85,B 0,C 180,E1 16904.265,E2 16904.265} C_VEL
LIN {X 0,Y 338.868,Z 809.795,A -85,B 0,C 180,E1 16907.402,E2 16907.402} C_VEL
LIN {X 0,Y 335.705,Z 826.401,A -85,B 0,C 180,E1 16912.765,E2 16912.765} C_VEL
LIN {X 0,Y 334.48,Z 842.558,A -85,B 0,C 180,E1 16917.43,E2 16917.43} C_VEL
LIN {X 0,Y 305.29,Z 898.404,A -85,B 0,C 180,E1 16924.308,E2 16924.308} C_VEL
LIN {X 0,Y 275.376,Z 944.717,A -85,B 0,C 180,E1 16934.811,E2 16934.811} C_VEL
LIN {X 0,Y 253.696,Z 977.025,A -85,B 0,C 180,E1 16948.775,E2 16948.775} C_VEL
LIN {X 0,Y 245.225,Z 992.677,A -85,B 0,C 180,E1 16961.878,E2 16961.878} C_VEL
LIN {X 0,Y 241.904,Z 998.559,A -85,B 0,C 180,E1 16973.419,E2 16973.419} C_VEL
LIN {X 0,Y 243.372,Z 995.566,A -85,B 0,C 180,E1 16988.544,E2 16988.544} C_VEL
LIN {X 0,Y 249.836,Z 980.78,A -85,B 0,C 180,E1 17003.024,E2 17003.024} C_VEL
LIN {X 0,Y 267.272,Z 950.395,A -85,B 0,C 180,E1 17017.424,E2 17017.424} C_VEL
LIN {X 0,Y 292.616,Z 906.342,A -85,B 0,C 180,E1 17028.523,E2 17028.523} C_VEL
LIN {X 0,Y 318.92,Z 851.389,A -85,B 0,C 180,E1 17036.116,E2 17036.116} C_VEL
LIN {X 0,Y 324.412,Z 834.324,A -85,B 0,C 180,E1 17038.07,E2 17038.07} C_VEL
LIN {X 0,Y 314.167,Z 800.294,A -85,B 0,C 180,E1 17047.56,E2 17047.56} C_VEL
LIN {X 0,Y 301.663,Z 773.041,A -85,B 0,C 180,E1 17058.697,E2 17058.697} C_VEL
LIN {X 0,Y 292.524,Z 757.287,A -85,B 0,C 180,E1 17070.17,E2 17070.17} C_VEL
LIN {X 0,Y 289.107,Z 751.501,A -85,B 0,C 180,E1 17079.304,E2 17079.304} C_VEL
LIN {X 0,Y 290.891,Z 752.104,A -85,B 0,C 180,E1 17092.204,E2 17092.204} C_VEL
LIN {X 0,Y 295.634,Z 758.609,A -85,B 0,C 180,E1 17100.1,E2 17100.1} C_VEL
LIN {X 0,Y 306.639,Z 778.344,A -85,B 0,C 180,E1 17111.382,E2 17111.382} C_VEL
LIN {X 0,Y 320.608,Z 810.673,A -85,B 0,C 180,E1 17122.359,E2 17122.359} C_VEL
LIN {X 0,Y 328.05,Z 838.92,A -85,B 0,C 180,E1 17129.074,E2 17129.074} C_VEL
LIN {X 0,Y 302.76,Z 898.541,A -85,B 0,C 180,E1 17135.266,E2 17135.266} C_VEL
LIN {X 0,Y 275.929,Z 948.953,A -85,B 0,C 180,E1 17144.916,E2 17144.916} C_VEL
LIN {X 0,Y 255.335,Z 985.524,A -85,B 0,C 180,E1 17157.66,E2 17157.66} C_VEL
LIN {X 0,Y 245.018,Z 1007.57,A -85,B 0,C 180,E1 17171.958,E2 17171.958} C_VEL
LIN {X 0,Y 243.146,Z 1016.177,A -85,B 0,C 180,E1 17184.626,E2 17184.626} C_VEL
LIN {X 0,Y 243.151,Z 1016.253,A -85,B 0,C 180,E1 17195.37,E2 17195.37} C_VEL
LIN {X 0,Y 245.812,Z 1006.025,A -85,B 0,C 180,E1 17209.848,E2 17209.848} C_VEL
LIN {X 0,Y 257.972,Z 982.203,A -85,B 0,C 180,E1 17224.625,E2 17224.625} C_VEL
LIN {X 0,Y 282.308,Z 943.203,A -85,B 0,C 180,E1 17237.506,E2 17237.506} C_VEL
LIN {X 0,Y 312.469,Z 892.061,A -85,B 0,C 180,E1 17246.707,E2 17246.707} C_VEL
LIN {X 0,Y 337.291,Z 838.959,A -85,B 0,C 180,E1 17252.377,E2 17252.377} C_VEL
LIN {X 0,Y 335.857,Z 820.085,A -85,B 0,C 180,E1 17259.538,E2 17259.538} C_VEL
LIN {X 0,Y 335.663,Z 815.494,A -85,B 0,C 180,E1 17265.636,E2 17265.636} C_VEL
LIN {X 0,Y 335.705,Z 826.401,A -85,B 0,C 180,E1 17272.765,E2 17272.765} C_VEL
LIN {X 0,Y 330.754,Z 842.737,A -85,B 0,C 180,E1 17275.666,E2 17275.666} C_VEL
LIN {X 0,Y 322.837,Z 860.478,A -85,B 0,C 180,E1 17277.825,E2 17277.825} C_VEL
LIN {X 0,Y 292.294,Z 912.565,A -85,B 0,C 180,E1 17285.466,E2 17285.466} C_VEL
LIN {X 0,Y 262.914,Z 954.565,A -85,B 0,C 180,E1 17296.803,E2 17296.803} C_VEL
LIN {X 0,Y 242.763,Z 983.701,A -85,B 0,C 180,E1 17312.138,E2 17312.138} C_VEL
LIN {X 0,Y 235.177,Z 997.138,A -85,B 0,C 180,E1 17327.958,E2 17327.958} C_VEL
LIN {X 0,Y 233.806,Z 998.862,A -85,B 0,C 180,E1 17341.258,E2 17341.258} C_VEL
LIN {X 0,Y 237.641,Z 991.003,A -85,B 0,C 180,E1 17355.286,E2 17355.286} C_VEL
LIN {X 0,Y 249.253,Z 968.934,A -85,B 0,C 180,E1 17370.874,E2 17370.874} C_VEL
LIN {X 0,Y 271.418,Z 933.33,A -85,B 0,C 180,E1 17383.748,E2 17383.748} C_VEL
LIN {X 0,Y 299.009,Z 884.259,A -85,B 0,C 180,E1 17393.362,E2 17393.362} C_VEL
LIN {X 0,Y 318.687,Z 838.21,A -85,B 0,C 180,E1 17398.868,E2 17398.868} C_VEL
LIN {X 0,Y 309.013,Z 804.462,A -85,B 0,C 180,E1 17408.75,E2 17408.75} C_VEL
LIN {X 0,Y 298.116,Z 779.588,A -85,B 0,C 180,E1 17419.415,E2 17419.415} C_VEL
LIN {X 0,Y 289.814,Z 764.167,A -85,B 0,C 180,E1 17430.944,E2 17430.944} C_VEL
LIN {X 0,Y 286.934,Z 758.057,A -85,B 0,C 180,E1 17443.056,E2 17443.056} C_VEL
LIN {X 0,Y 291.796,Z 763.204,A -85,B 0,C 180,E1 17457.544,E2 17457.544} C_VEL
LIN {X 0,Y 301.693,Z 782.46,A -85,B 0,C 180,E1 17469.588,E2 17469.588} C_VEL
LIN {X 0,Y 314.286,Z 811.544,A -85,B 0,C 180,E1 17480.379,E2 17480.379} C_VEL
LIN {X 0,Y 322.543,Z 841.521,A -85,B 0,C 180,E1 17488.105,E2 17488.105} C_VEL
LIN {X 0,Y 297.074,Z 899.333,A -85,B 0,C 180,E1 17494.201,E2 17494.201} C_VEL
LIN {X 0,Y 269.171,Z 949.748,A -85,B 0,C 180,E1 17504.038,E2 17504.038} C_VEL
LIN {X 0,Y 247.226,Z 986.826,A -85,B 0,C 180,E1 17517.51,E2 17517.51} C_VEL
LIN {X 0,Y 237.235,Z 1007.182,A -85,B 0,C 180,E1 17531.344,E2 17531.344} C_VEL
LIN {X 0,Y 235.146,Z 1015.856,A -85,B 0,C 180,E1 17544.443,E2 17544.443} C_VEL
LIN {X 0,Y 235.151,Z 1015.967,A -85,B 0,C 180,E1 17555.554,E2 17555.554} C_VEL
LIN {X 0,Y 238.026,Z 1005.782,A -85,B 0,C 180,E1 17570.526,E2 17570.526} C_VEL
LIN {X 0,Y 251.455,Z 981.586,A -85,B 0,C 180,E1 17585.936,E2 17585.936} C_VEL
LIN {X 0,Y 277.749,Z 941.845,A -85,B 0,C 180,E1 17599.145,E2 17599.145} C_VEL
LIN {X 0,Y 309.122,Z 890.9,A -85,B 0,C 180,E1 17608.202,E2 17608.202} C_VEL
LIN {X 0,Y 332.62,Z 843.434,A -85,B 0,C 180,E1 17613.276,E2 17613.276} C_VEL
LIN {X 0,Y 332.085,Z 826.675,A -85,B 0,C 180,E1 17619.993,E2 17619.993} C_VEL
LIN {X 0,Y 332.022,Z 822.663,A -85,B 0,C 180,E1 17625.475,E2 17625.475} C_VEL
LIN {X 0,Y 331.399,Z 833.974,A -85,B 0,C 180,E1 17632.798,E2 17632.798} C_VEL
LIN {X 0,Y 330.754,Z 842.737,A -85,B 0,C 180,E1 17635.666,E2 17635.666} C_VEL
LIN {X 0,Y 325.904,Z 852.164,A -85,B 0,C 180,E1 17636.368,E2 17636.368} C_VEL
LIN {X 0,Y 318.822,Z 862.775,A -85,B 0,C 180,E1 17636.666,E2 17636.666} C_VEL
LIN {X 0,Y 286.079,Z 915.656,A -85,B 0,C 180,E1 17644.598,E2 17644.598} C_VEL
LIN {X 0,Y 255.934,Z 956.374,A -85,B 0,C 180,E1 17656.045,E2 17656.045} C_VEL
LIN {X 0,Y 235.104,Z 984.597,A -85,B 0,C 180,E1 17671.641,E2 17671.641} C_VEL
LIN {X 0,Y 228.001,Z 996.614,A -85,B 0,C 180,E1 17685.665,E2 17685.665} C_VEL
LIN {X 0,Y 225.589,Z 999.349,A -85,B 0,C 180,E1 17699.701,E2 17699.701} C_VEL
LIN {X 0,Y 229.086,Z 992.788,A -85,B 0,C 180,E1 17713.965,E2 17713.965} C_VEL
LIN {X 0,Y 240.072,Z 972.71,A -85,B 0,C 180,E1 17730.002,E2 17730.002} C_VEL
LIN {X 0,Y 262.807,Z 937.684,A -85,B 0,C 180,E1 17743.782,E2 17743.782} C_VEL
LIN {X 0,Y 290.738,Z 890.33,A -85,B 0,C 180,E1 17753.727,E2 17753.727} C_VEL
LIN {X 0,Y 312.877,Z 841.635,A -85,B 0,C 180,E1 17759.814,E2 17759.814} C_VEL
LIN {X 0,Y 304.574,Z 810.201,A -85,B 0,C 180,E1 17769.403,E2 17769.403} C_VEL
LIN {X 0,Y 293.985,Z 785.135,A -85,B 0,C 180,E1 17780.743,E2 17780.743} C_VEL
LIN {X 0,Y 286.547,Z 768.789,A -85,B 0,C 180,E1 17793.649,E2 17793.649} C_VEL
LIN {X 0,Y 285.579,Z 766.311,A -85,B 0,C 180,E1 17809.248,E2 17809.248} C_VEL
LIN {X 0,Y 290.128,Z 772.686,A -85,B 0,C 180,E1 17818.842,E2 17818.842} C_VEL
LIN {X 0,Y 300.149,Z 793.046,A -85,B 0,C 180,E1 17830.893,E2 17830.893} C_VEL
LIN {X 0,Y 311.848,Z 823.878,A -85,B 0,C 180,E1 17841.741,E2 17841.741} C_VEL
LIN {X 0,Y 316.641,Z 845.31,A -85,B 0,C 180,E1 17847.201,E2 17847.201} C_VEL
LIN {X 0,Y 290.806,Z 901.307,A -85,B 0,C 180,E1 17853.284,E2 17853.284} C_VEL
LIN {X 0,Y 262.485,Z 950.527,A -85,B 0,C 180,E1 17863.117,E2 17863.117} C_VEL
LIN {X 0,Y 239.118,Z 988.127,A -85,B 0,C 180,E1 17877.351,E2 17877.351} C_VEL
LIN {X 0,Y 228.721,Z 1008.621,A -85,B 0,C 180,E1 17892.626,E2 17892.626} C_VEL
LIN {X 0,Y 227.136,Z 1015.534,A -85,B 0,C 180,E1 17904.246,E2 17904.246} C_VEL
LIN {X 0,Y 227.141,Z 1015.682,A -85,B 0,C 180,E1 17915.75,E2 17915.75} C_VEL
LIN {X 0,Y 230.29,Z 1005.553,A -85,B 0,C 180,E1 17931.249,E2 17931.249} C_VEL
LIN {X 0,Y 244.892,Z 981.297,A -85,B 0,C 180,E1 17947.17,E2 17947.17} C_VEL
LIN {X 0,Y 273.119,Z 941.032,A -85,B 0,C 180,E1 17960.709,E2 17960.709} C_VEL
LIN {X 0,Y 306.247,Z 889.46,A -85,B 0,C 180,E1 17969.778,E2 17969.778} C_VEL
LIN {X 0,Y 328.032,Z 847.105,A -85,B 0,C 180,E1 17974.438,E2 17974.438} C_VEL
LIN {X 0,Y 328.185,Z 832.017,A -85,B 0,C 180,E1 17981.431,E2 17981.431} C_VEL
LIN {X 0,Y 328.049,Z 830.774,A -85,B 0,C 180,E1 17986.661,E2 17986.661} C_VEL
LIN {X 0,Y 326.702,Z 843.11,A -85,B 0,C 180,E1 17993.364,E2 17993.364} C_VEL
LIN {X 0,Y 324.42,Z 852.165,A -85,B 0,C 180,E1 17995.579,E2 17995.579} C_VEL
LIN {X 0,Y 318.822,Z 862.775,A -85,B 0,C 180,E1 17996.666,E2 17996.666} C_VEL
LIN {X 0,Y 299.51,Z 890.449,A -85,B 0,C 180,E1 17998.703,E2 17998.703} C_VEL
LIN {X 0,Y 265.609,Z 937.618,A -85,B 0,C 180,E1 18008.248,E2 18008.248} C_VEL
LIN {X 0,Y 236.624,Z 973.552,A -85,B 0,C 180,E1 18022.68,E2 18022.68} C_VEL
LIN {X 0,Y 222.642,Z 992.586,A -85,B 0,C 180,E1 18038.386,E2 18038.386} C_VEL
LIN {X 0,Y 217.741,Z 999.666,A -85,B 0,C 180,E1 18053.673,E2 18053.673} C_VEL
LIN {X 0,Y 219.452,Z 996.651,A -85,B 0,C 180,E1 18069.09,E2 18069.09} C_VEL
LIN {X 0,Y 227.693,Z 981.311,A -85,B 0,C 180,E1 18085.549,E2 18085.549} C_VEL
LIN {X 0,Y 247.617,Z 951.656,A -85,B 0,C 180,E1 18100.573,E2 18100.573} C_VEL
LIN {X 0,Y 276.352,Z 907.103,A -85,B 0,C 180,E1 18112.183,E2 18112.183} C_VEL
LIN {X 0,Y 305.228,Z 851.849,A -85,B 0,C 180,E1 18119.797,E2 18119.797} C_VEL
LIN {X 0,Y 307.107,Z 844.786,A -85,B 0,C 180,E1 18120.856,E2 18120.856} C_VEL
LIN {X 0,Y 298.969,Z 812.922,A -85,B 0,C 180,E1 18131.162,E2 18131.162} C_VEL
LIN {X 0,Y 289.41,Z 789.031,A -85,B 0,C 180,E1 18142.88,E2 18142.88} C_VEL
LIN {X 0,Y 282.988,Z 775.568,A -85,B 0,C 180,E1 18156.251,E2 18156.251} C_VEL
LIN {X 0,Y 283.231,Z 773.925,A -85,B 0,C 180,E1 18169.158,E2 18169.158} C_VEL
LIN {X 0,Y 287.3,Z 779.924,A -85,B 0,C 180,E1 18178.452,E2 18178.452} C_VEL
LIN {X 0,Y 296.314,Z 799.398,A -85,B 0,C 180,E1 18190.289,E2 18190.289} C_VEL
LIN {X 0,Y 306.797,Z 828.774,A -85,B 0,C 180,E1 18200.975,E2 18200.975} C_VEL
LIN {X 0,Y 310.898,Z 848.791,A -85,B 0,C 180,E1 18206.239,E2 18206.239} C_VEL
LIN {X 0,Y 282.558,Z 907.08,A -85,B 0,C 180,E1 18212.915,E2 18212.915} C_VEL
LIN {X 0,Y 253.702,Z 954.278,A -85,B 0,C 180,E1 18223.025,E2 18223.025} C_VEL
